60200:
	IF NOT Robot._DI1.Done THEN
		IF _bTargetIsA THEN
			Robot.M_StartMoveBoxToRoundBelt_ClampA(
				CarrierSelect := Info.ClampA_Setting.RoundBeltSetting.ReloadCarrier,
				A2_Sensor := A2_Sensor, A3_Sensor := A3_Sensor,
				RoundBeltSafe := CarrierReady_1st);
		ELSE
			Robot.M_StartMoveBoxToRoundBelt_ClampB(
				CarrierSelect := Info.ClampB_Setting.RoundBeltSetting.ReloadCarrier,
				A2_Sensor := A2_Sensor, A3_Sensor := A3_Sensor,
				RoundBeltSafe := CarrierReady_1st);
		END_IF
	ELSE
		// 圓帶放盒不記數 (非倉儲操作)
		tonTimeOut.IN := FALSE;
		uiExecutingStep := 60300;
	END_IF
	tonTimeOut.IN := TRUE;
	IF tonTimeOut.Q THEN uiResumeStep := 60200; _Abort := TRUE; tonTimeOut.IN := FALSE; END_IF

60300:
	// 釋放圓帶資源 + 清除手臂命令 → 三路分派:
	// 1. buffer > 0: 先去 90000 逆序還原 buffer 盒子 (還原完再由 90010 判斷跳轉)
	// 2. _nAfterPlaceStep > 0: C3/C4 的下一輪入口 (如 3250/3350)
	// 3. 否則: 99000 全部完成
	DAS_CoreSys.MachineControl.fbAllocateArea.M_ResetReloadRoundBeltAction();
	DAS_CoreSys.MachineControl.fbAllocateArea.M_ReleaseRoundBeltAccess(ControlAccess := E_RoundBeltControlAccess.FanucRobot);
	Robot.M_ResetAllCommand();
	IF NOT Robot._DI1.Done THEN
		IF _nBufferCount > 0 THEN
			uiExecutingStep := 90000;
		ELSIF _nAfterPlaceStep > 0 THEN
			uiExecutingStep := _nAfterPlaceStep;
			_nAfterPlaceStep := 0;
		ELSE
			uiExecutingStep := 99000;
		END_IF
	END_IF

// ========== 80000: 雙爪放盒到圓帶 (A 爪先放, B 爪後放) ==========
// 80000: 清除命令 + 立即進入圓帶流程 (不等手臂空閒，並行啟動)
// 81000: 雙爪放圓帶主迴圈 (子步序 uiPlaceBothStep):
//   0:  取得圓帶存取權
//   10: 移動圓帶到 A 爪站位 → 等待到位
//   11: 等待 A 爪載具 sensor 確認 (A2/A3) → 再次取得圓帶存取權
//   20: 等待 Robot Notification (A 爪放完) → Reset 圓帶動作
//   30: 移動圓帶到 B 爪站位
//   40: 等待 B 爪載具到位
//   99: 等待手臂完成
// 81080: 釋放圓帶存取權 + 清除命令 → buffer 還原或完成
80000:
	// 圓帶先動 — 不等手臂完全空閒，手臂清除與圓帶移動並行
	WareHouse.M_ResetReloadBox();
	Robot.M_ResetAllCommand();
	uiExecutingStep := 81000;

81000:
	// ── 子步序: 圓帶側與手臂側並行協調 ──
	// 圓帶側 (uiPlaceBothStep): 依序移到 A站位→確認載具→等A放完→移到 B站位→確認載具
	// 手臂側 (下方 M_StartMoveBoxToRoundBelt_Both): 每 cycle 持續呼叫，根據 CarrierReady 旗標推進
	CASE uiPlaceBothStep OF
	0:
		// 初始化: 取得圓帶控制權，立即開始移動
		CarrierReady_1st := FALSE;
		CarrierReady_2nd := FALSE;
		DAS_CoreSys.MachineControl.fbAllocateArea.M_GetRoundBeltAccess(ControlAccess := E_RoundBeltControlAccess.FanucRobot);
		uiPlaceBothStep := 10;
	10:
		// 圓帶移到 A 爪站位，等待到位 (與手臂清除並行)
		DAS_CoreSys.MachineControl.fbAllocateArea.M_StartReloadRoundBeltAtion(ReloadStation := Info.ClampA_Setting.RoundBeltSetting.Station);
		IF RoundBelt.xDone THEN
			DAS_CoreSys.MachineControl.fbAllocateArea.M_ResetReloadRoundBeltAction();
			DAS_CoreSys.MachineControl.fbAllocateArea.M_ReleaseRoundBeltAccess(ControlAccess := E_RoundBeltControlAccess.FanucRobot);
			CarrierReady_1st := TRUE;	// → 手臂開始 A 爪放盒
			uiPlaceBothStep := 11;
		END_IF
		IF RoundBelt.xError THEN
			_Error := TRUE;
			DAS_CoreSys.MachineControl.fbAllocateArea.M_ResetReloadRoundBeltAction();
			strStatus := 'FB_WareHouseInnerPickToRoundBelt Step 81000: RoundBelt error';
		END_IF
	11:
		// 等待 A 爪對應的載具 sensor 偵測到位 (確認載具已在手臂放盒範圍內)
		// A2 載具用 A2_Sensor 確認, A3 載具用 A3_Sensor 確認
		IF ((Info.ClampA_Setting.RoundBeltSetting.ReloadCarrier = E_ReloadRoundBelt_PlaceAddress.A2) AND A2_Sensor) OR
			((Info.ClampA_Setting.RoundBeltSetting.ReloadCarrier = E_ReloadRoundBelt_PlaceAddress.A3) AND A3_Sensor) THEN
			// 載具到位 → 重新取得圓帶權限 (step 10 釋放過)，準備等手臂放完後移到 B 站位
			DAS_CoreSys.MachineControl.fbAllocateArea.M_GetRoundBeltAccess(ControlAccess := E_RoundBeltControlAccess.FanucRobot);
			uiPlaceBothStep := 20;
		END_IF
	20:
		// 等待手臂 Notification = A 爪放盒完成信號 (手臂程式中途發出，不等全部結束)
		IF Robot._DI1.Notification THEN
			DAS_CoreSys.MachineControl.fbAllocateArea.M_ResetReloadRoundBeltAction();
			// 確認圓帶不在 Done 狀態 (已被 Reset)，才開始移到 B 站位
			IF NOT RoundBelt.xDone THEN
				uiPlaceBothStep := 30;
			END_IF
		END_IF
	30:
		// 圓帶移到 B 爪站位
		DAS_CoreSys.MachineControl.fbAllocateArea.M_GetRoundBeltAccess(ControlAccess := E_RoundBeltControlAccess.FanucRobot);
		DAS_CoreSys.MachineControl.fbAllocateArea.M_StartReloadRoundBeltAtion(ReloadStation := Info.ClampB_Setting.RoundBeltSetting.Station);
		uiPlaceBothStep := 40;
	40:
		// 等待 B 爪站位到位
		IF RoundBelt.xDone THEN
			DAS_CoreSys.MachineControl.fbAllocateArea.M_ResetReloadRoundBeltAction();
			CarrierReady_2nd := TRUE;	// → 手臂開始 B 爪放盒
			uiPlaceBothStep := 99;
		END_IF
		IF RoundBelt.xError THEN
			_Error := TRUE;
			DAS_CoreSys.MachineControl.fbAllocateArea.M_ResetReloadRoundBeltAction();
			strStatus := 'FB_WareHouseInnerPickToRoundBelt Step 81000: RoundBelt error';
		END_IF
	99: // 圓帶側完成，等待手臂側 Done
	END_CASE

	// 手臂側: 每 cycle 持續呼叫，手臂內部根據 CarrierReady 旗標推進雙爪放盒流程
	IF NOT Robot._DI1.Done THEN
		Robot.M_StartMoveBoxToRoundBelt_Both(
			CarrierSelect_ClampA := Info.ClampA_Setting.RoundBeltSetting.ReloadCarrier,
			CarrierSelect_ClampB := Info.ClampB_Setting.RoundBeltSetting.ReloadCarrier,
			A2_Sensor := A2_Sensor, A3_Sensor := A3_Sensor,
			RoundBeltSafe_1st := CarrierReady_1st,
			RoundBeltSafe_2nd := CarrierReady_2nd);
	ELSE
		// 圓帶放盒不記數 (非倉儲操作)
		tonTimeOut.IN := FALSE;
		uiExecutingStep := 81080;
	END_IF
	tonTimeOut.IN := TRUE;
	IF tonTimeOut.Q THEN uiResumeStep := 81000; _Abort := TRUE; tonTimeOut.IN := FALSE; END_IF

81080:
	DAS_CoreSys.MachineControl.fbAllocateArea.M_ResetReloadRoundBeltAction();
	DAS_CoreSys.MachineControl.fbAllocateArea.M_ReleaseRoundBeltAccess(ControlAccess := E_RoundBeltControlAccess.FanucRobot);
	Robot.M_ResetAllCommand();
	IF NOT Robot._DI1.Done THEN
		IF _nBufferCount > 0 THEN
			uiExecutingStep := 90000;		// 有 buffer 要還原
		ELSIF _nAfterPlaceStep > 0 THEN
			uiExecutingStep := _nAfterPlaceStep;	// C3/C4 跳轉到下一輪
			_nAfterPlaceStep := 0;
		ELSE
			uiExecutingStep := 99000;		// 完成
		END_IF
	END_IF

// ========== 90000: Buffer 盒子逆序還原 ==========
// 將之前搬到 buffer 的盒子，逆序 (後進先出) 放回倉儲
// 雙爪路徑: 一次從 buffer 取兩個 → 依序放回倉儲
// 單爪路徑: 剩一個時用目標爪處理
90000:
	_nBufferStep := _nBufferCount;
	BoxReady_1st := FALSE;
	BoxReady_2nd := FALSE;
	uiExecutingStep := 90005;

90005:
	IF _nBufferStep < 1 THEN
		// buffer 還原完成 → 檢查是否有下一輪跳轉 (C3/C4)
		IF _nAfterPlaceStep > 0 THEN
			uiExecutingStep := _nAfterPlaceStep;
			_nAfterPlaceStep := 0;
		ELSE
			uiExecutingStep := 99000;
		END_IF
	ELSIF _nBufferStep >= 2 THEN
		// 剩 2 個以上: 雙爪一次還原兩個
		uiExecutingStep := 90010;
	ELSE
		// 剩 1 個: 單爪還原
		uiExecutingStep := 90040;
	END_IF

// ===== 雙爪 buffer 還原路徑 =====
// Step 1: 雙爪從 buffer 取兩個盒子
90010:
	IF NOT Robot._DI1.Done THEN
		IF _bTargetIsA THEN
			Robot.M_StartRobotAbsMove(
				GetBox := TRUE, UseClampA := TRUE, UseClampB := TRUE,
				Area := E_RobotArea.BufferArea,
				ClampA_Address := _nBufferStep, ClampB_Address := _nBufferStep - 1,
				BoxReady_1 := TRUE, BoxReady_2 := TRUE);
		ELSE
			Robot.M_StartRobotAbsMove(
				GetBox := TRUE, UseClampA := TRUE, UseClampB := TRUE,
				Area := E_RobotArea.BufferArea,
				ClampA_Address := _nBufferStep - 1, ClampB_Address := _nBufferStep,
				BoxReady_1 := TRUE, BoxReady_2 := TRUE);
		END_IF
	ELSE
		// buffer 取盒不記數 (非倉儲操作)
		tonTimeOut.IN := FALSE;
		uiExecutingStep := 90015;
	END_IF
	tonTimeOut.IN := TRUE;
	IF tonTimeOut.Q THEN uiResumeStep := 90010; _Abort := TRUE; tonTimeOut.IN := FALSE; END_IF

90015:
	Robot.M_ResetAllCommand();
	IF NOT Robot._DI1.Done THEN
		BoxReady_1st := FALSE;
		BoxReady_2nd := FALSE;
		uiExecutingStep := 90020;
	END_IF

// Step 2: 目標爪放回倉儲 (buffer 高位, LIFO 先還原)
90020:
	IF NOT Robot._DI1.Done THEN
		IF _bTargetIsA THEN
			WareHouse.M_StartFeedInBox(WareHouseSelect := _wsA, WarehouseCoordinates := _coordsA);
			IF WareHouse.bFeedInBox_Completed THEN BoxReady_1st := TRUE; END_IF
			Robot.M_StartWareHousePlaceBox_ClampA(WareHouseSelect := _wsA, Info := _coordsA, BoxReady_1st := BoxReady_1st);
		ELSE
			WareHouse.M_StartFeedInBox(WareHouseSelect := _wsB, WarehouseCoordinates := _coordsB);
			IF WareHouse.bFeedInBox_Completed THEN BoxReady_2nd := TRUE; END_IF
			Robot.M_StartWareHousePlaceBox_ClampB(WareHouseSelect := _wsB, Info := _coordsB, BoxReady_2nd := BoxReady_2nd);
		END_IF
	ELSE
		// Place 完成通知: 目標爪放回倉儲 (buffer 高位)
		IF ActionIndex < 40 THEN
			IF _bTargetIsA THEN
				ActionRecords[ActionIndex].WareHouse := _wsA; ActionRecords[ActionIndex].Layer := _coordsA.Layer; ActionRecords[ActionIndex].Slide := _coordsA.Slide; ActionRecords[ActionIndex].Clamp := 0;
			ELSE
				ActionRecords[ActionIndex].WareHouse := _wsB; ActionRecords[ActionIndex].Layer := _coordsB.Layer; ActionRecords[ActionIndex].Slide := _coordsB.Slide; ActionRecords[ActionIndex].Clamp := 1;
			END_IF
			ActionRecords[ActionIndex].IsPick := FALSE;
			ActionIndex := ActionIndex + 1;
		END_IF
		tonTimeOut.IN := FALSE;
		uiExecutingStep := 90025;
	END_IF
	tonTimeOut.IN := TRUE;
	IF tonTimeOut.Q THEN uiResumeStep := 90020; _Abort := TRUE; tonTimeOut.IN := FALSE; END_IF

90025:
	Robot.M_ResetAllCommand();
	WareHouse.M_ResetFeedInBox();
	IF NOT Robot._DI1.Done THEN
		BoxReady_1st := FALSE;
		BoxReady_2nd := FALSE;
		uiExecutingStep := 90030;
	END_IF

// Step 3: 協助爪放回倉儲 (buffer 低位)
90030:
	IF NOT Robot._DI1.Done THEN
		IF _bTargetIsA THEN
			WareHouse.M_StartFeedInBox(WareHouseSelect := _wsA, WarehouseCoordinates := _coordsA);
			IF WareHouse.bFeedInBox_Completed THEN BoxReady_2nd := TRUE; END_IF
			Robot.M_StartWareHousePlaceBox_ClampB(WareHouseSelect := _wsA, Info := _coordsA, BoxReady_2nd := BoxReady_2nd);
		ELSE
			WareHouse.M_StartFeedInBox(WareHouseSelect := _wsB, WarehouseCoordinates := _coordsB);
			IF WareHouse.bFeedInBox_Completed THEN BoxReady_1st := TRUE; END_IF
			Robot.M_StartWareHousePlaceBox_ClampA(WareHouseSelect := _wsB, Info := _coordsB, BoxReady_1st := BoxReady_1st);
		END_IF
	ELSE
		// Place 完成通知: 協助爪放回倉儲 (buffer 低位)
		IF ActionIndex < 40 THEN
			IF _bTargetIsA THEN
				ActionRecords[ActionIndex].WareHouse := _wsA; ActionRecords[ActionIndex].Layer := _coordsA.Layer; ActionRecords[ActionIndex].Slide := _coordsA.Slide; ActionRecords[ActionIndex].Clamp := 1;
			ELSE
				ActionRecords[ActionIndex].WareHouse := _wsB; ActionRecords[ActionIndex].Layer := _coordsB.Layer; ActionRecords[ActionIndex].Slide := _coordsB.Slide; ActionRecords[ActionIndex].Clamp := 0;
			END_IF
			ActionRecords[ActionIndex].IsPick := FALSE;
			ActionIndex := ActionIndex + 1;
		END_IF
		tonTimeOut.IN := FALSE;
		uiExecutingStep := 90035;
	END_IF
	tonTimeOut.IN := TRUE;
	IF tonTimeOut.Q THEN uiResumeStep := 90030; _Abort := TRUE; tonTimeOut.IN := FALSE; END_IF

90035:
	Robot.M_ResetAllCommand();
	WareHouse.M_ResetFeedInBox();
	IF NOT Robot._DI1.Done THEN
		BoxReady_1st := FALSE;
		BoxReady_2nd := FALSE;
		_nBufferStep := _nBufferStep - 2;
		uiExecutingStep := 90005;
	END_IF

// ===== 單爪 buffer 還原路徑 (剩一個) =====
90040:
	IF NOT Robot._DI1.Done THEN
		IF _bTargetIsA THEN
			Robot.M_StartRobotAbsMove(
				GetBox := TRUE, UseClampA := TRUE, UseClampB := FALSE,
				Area := E_RobotArea.BufferArea,
				ClampA_Address := _nBufferStep, ClampB_Address := 0,
				BoxReady_1 := TRUE, BoxReady_2 := FALSE);
		ELSE
			Robot.M_StartRobotAbsMove(
				GetBox := TRUE, UseClampA := FALSE, UseClampB := TRUE,
				Area := E_RobotArea.BufferArea,
				ClampA_Address := 0, ClampB_Address := _nBufferStep,
				BoxReady_1 := FALSE, BoxReady_2 := TRUE);
		END_IF
	ELSE
		// buffer 取盒不記數 (非倉儲操作)
		tonTimeOut.IN := FALSE;
		uiExecutingStep := 90045;
	END_IF
	tonTimeOut.IN := TRUE;
	IF tonTimeOut.Q THEN uiResumeStep := 90040; _Abort := TRUE; tonTimeOut.IN := FALSE; END_IF

90045:
	Robot.M_ResetAllCommand();
	IF NOT Robot._DI1.Done THEN
		BoxReady_1st := FALSE;
		BoxReady_2nd := FALSE;
		uiExecutingStep := 90050;
	END_IF

90050:
	IF NOT Robot._DI1.Done THEN
		IF _bTargetIsA THEN
			WareHouse.M_StartFeedInBox(WareHouseSelect := _wsA, WarehouseCoordinates := _coordsA);
			IF WareHouse.bFeedInBox_Completed THEN BoxReady_1st := TRUE; END_IF
			Robot.M_StartWareHousePlaceBox_ClampA(WareHouseSelect := _wsA, Info := _coordsA, BoxReady_1st := BoxReady_1st);
		ELSE
			WareHouse.M_StartFeedInBox(WareHouseSelect := _wsB, WarehouseCoordinates := _coordsB);
			IF WareHouse.bFeedInBox_Completed THEN BoxReady_2nd := TRUE; END_IF
			Robot.M_StartWareHousePlaceBox_ClampB(WareHouseSelect := _wsB, Info := _coordsB, BoxReady_2nd := BoxReady_2nd);
		END_IF
	ELSE
		// Place 完成通知: 放回倉儲 (buffer 逆序還原)
		IF ActionIndex < 40 THEN
			IF _bTargetIsA THEN
				ActionRecords[ActionIndex].WareHouse := _wsA; ActionRecords[ActionIndex].Layer := _coordsA.Layer; ActionRecords[ActionIndex].Slide := _coordsA.Slide; ActionRecords[ActionIndex].Clamp := 0;
			ELSE
				ActionRecords[ActionIndex].WareHouse := _wsB; ActionRecords[ActionIndex].Layer := _coordsB.Layer; ActionRecords[ActionIndex].Slide := _coordsB.Slide; ActionRecords[ActionIndex].Clamp := 1;
			END_IF
			ActionRecords[ActionIndex].IsPick := FALSE;
			ActionIndex := ActionIndex + 1;
		END_IF
		tonTimeOut.IN := FALSE;
		uiExecutingStep := 90055;
	END_IF
	tonTimeOut.IN := TRUE;
	IF tonTimeOut.Q THEN uiResumeStep := 90050; _Abort := TRUE; tonTimeOut.IN := FALSE; END_IF

90055:
	Robot.M_ResetAllCommand();
	WareHouse.M_ResetFeedInBox();
	IF NOT Robot._DI1.Done THEN
		BoxReady_1st := FALSE;
		BoxReady_2nd := FALSE;
		_nBufferStep := _nBufferStep - 1;
		uiExecutingStep := 90005;
	END_IF

// ========== 99000: 流程完成 → 等待 C# 讀取動作紀錄 ==========
99000:
	DAS_CoreSys.MachineControl.fbAllocateArea.M_ResetReloadRoundBeltAction();
	DAS_CoreSys.MachineControl.fbAllocateArea.M_ReleaseRoundBeltAccess(ControlAccess := E_RoundBeltControlAccess.FanucRobot);
	FeedBack := TRUE;
	uiExecutingStep := 99100;

// Step 99100: 等待 C# 確認讀取完成 (5 秒逾時保護)
99100:
	//tonReadComplete(IN := TRUE, PT := T#15S);
	tonReadComplete.IN := true;
	IF ReadComplete THEN
		FeedBack := FALSE;
		tonReadComplete.IN := FALSE;
		Status := 'FB_WareHouseInnerPickToRoundBelt Step 99100: Process completed';
		_Executed := TRUE;
	ELSIF tonReadComplete.Q THEN
		// C# 讀取逾時 → Abort + 設 resume 回 99100，Reset 後可續做
		tonReadComplete.IN := FALSE;
		strStatus := 'FB_WareHouseInnerPickToRoundBelt Step 99100: ReadComplete timeout (C# did not respond within 5s)';
		_UniqueErrorCode := 'E_READ_COMPLETE_TIMEOUT';
		uiResumeStep := 99100;
		_Abort := TRUE;
	END_IF

END_CASE

// 狀態轉換判斷 (每 cycle 在 CASE 之後檢查)
// 優先順序: 完成 > 外部取消 > 中止(逾時) > 錯誤
// _Executed: 由 step 99000 設定，需等 Robot.Halt 解除才實際轉換 (避免手臂急停中換狀態)
// NOT Execute: 外部 (Batch FB 或 HMI) 取消 Execute，直接進入 RESETTING
// _Abort: 由逾時或內部異常設定，進入 ABORTING 清理手臂/倉儲資源
// _Error: 由命令驗證失敗或圓帶錯誤設定，進入 STATE_ERROR 顯示錯誤
IF _Executed AND NOT Robot.Halt THEN
	eState := STATE_DONE;
ELSIF NOT Execute THEN
	eState := STATE_RESETTING;
ELSIF Abort OR _Abort THEN
	eState := STATE_ABORTING;
ELSIF _Error THEN
	eState := STATE_ERROR;
END_IF
END_METHOD

// 重置狀態 — 釋放所有資源 (圓帶/倉儲/手臂)，清除爪動作旗標
// 如果有恢復旗標 (_bRetry)，回到 STATE_EXECUTING 的中斷步序
METHOD M_STATE_RESETTING
VAR_INPUT
END_VAR
// Done := false 更改到Dormant 清除確保，上位檢查到done 後可以直接下Execute

CASE uiResettingStep OF
0:
	// 清除動作紀錄 + 握手旗標
	MEMSET(ADR(ActionRecords), 0, SIZEOF(ActionRecords));
	ActionIndex := 0;
	FeedBack := FALSE;

	// 釋放所有外部資源 → 圓帶/倉儲/手臂回到初始狀態
	DAS_CoreSys.MachineControl.fbAllocateArea.M_ResetReloadRoundBeltAction();
	DAS_CoreSys.MachineControl.fbAllocateArea.M_ReleaseRoundBeltAccess(ControlAccess := E_RoundBeltControlAccess.FanucRobot);
	WareHouse.M_ResetReloadBox();
	WareHouse.M_ResetFeedInBox();
	Robot.M_ResetAllCommand();

	// 清除內部狀態
	tonTimeOut.IN := FALSE;
	tonReadComplete.IN := FALSE;
	strStatus := '';
	_UniqueErrorCode := '0';

//	IF _bRetry THEN
//		_bRetry := FALSE;
//		eState := STATE_EXECUTING;
//		RETURN;
//	END_IF
	uiResettingStep := 100;
100:
//	Done := FALSE;
//	Busy := FALSE;
	_ResetCompleted := TRUE;
END_CASE

IF _ResetCompleted THEN
	eState := STATE_DORMANT;
END_IF
END_METHOD

END_FUNCTION_BLOCK

// ---- Library/20_MachineUnits/21_StorageArea/Service_Robot/FB_WareHouseInnerPickToRoundBeltBatch.TcPOU
// ═══════════════════════════════════════════════════════════════════════════
// FB_WareHouseInnerPickToRoundBeltBatch
// 倉儲內層取盒放圓帶 — 批次服務 FB
// ═══════════════════════════════════════════════════════════════════════════
//
// 【用途】
// 管理最多 40 筆「從倉儲內層取盒放上圓帶」流程,每筆由 FB_WareHouseInnerPickToRoundBelt
// 逐筆執行。批次流程由 C# HMI 透過 ADS 寫入 BatchInfo 結構觸發,PLC 端負責
// 驗證資料、迭代處理、handshake 同步動作紀錄給 C#。
//
// 【設計模式】
// 參照 FB_AllocateMoveAutoBatchMode,以「單筆 FB 內嵌 + 批次迭代」架構:
//   1. 收到 Execute → 驗證整批資料安全 (M_ValidateBatchData)
//   2. 迭代 FlowInfo[0..NrOfFlow-1]
//   3. 跳過無效項 (ID = -1 或 A/B 爪皆 NoWork)
//   4. 對每筆有效流程配置並啟動 fbSingleFlow,等其完成/失敗
//   5. 完成後記錄 WorkedID 供 HMI/C# 回報
//   6. 跨迭代 handshake 清理,確保 C# 看到每筆 FeedBack 上升緣
//
// 【FeedBack / ReadComplete 握手協定】(關鍵,跨迭代正確性依賴)
// 每筆 fbSingleFlow 完成時:
//   PLC:   step 99000 → FeedBack := TRUE (通知 C# 陣列可讀)
//   C#:    收到 FeedBack=TRUE → 讀 ActionRecords → set ReadComplete=TRUE
//   PLC:   step 99100 看 ReadComplete=TRUE → 清 FeedBack → 進 DONE
//   C#:    應在看到 FeedBack=FALSE 時清 ReadComplete=FALSE (維持協定)
// 本 Batch FB 為了防 C# 忘記清 ReadComplete 造成下一迭代 skip handshake,
// 在 Step 100 (新迭代開始) 與 Step 300 (迭代結束) 強制清 BatchInfo.ReadComplete。
//
// 【資料安全約束】
// M_ValidateBatchData 在 Step 0 首次進入時呼叫,檢查:
//   - 每個 Work clamp 的 Station 不可為 Undefined
//   - 所有 Work clamp 的 (Station, ReloadCarrier) 不可重複 (同 flow A/B 兩爪也算)
// 違規 → Error + uiResumeStep:=0 (不可續做,需 C# 修正資料重來)
//
// 【Resume / Pause】
// Resume: 錯誤/逾時後 C# 按 Reset → RESETTING 等 fbSingleFlow 回 DORMANT
//         → 若 _bRetry 直接回 EXECUTING 從 uiResumeStep 繼續
//         uiResumeStep 映射固定為 100 (重新配置+啟動 fbSingleFlow),因 abort
//         過程會清掉 fbSingleFlow 內部狀態,不能回原 step 200
// Pause:  僅在「迭代邊界」生效 (step 0 或 310),不中斷單筆流程
//         危險區段 (100~300) 繼續跑到下個邊界才凍結
//
// Create Date : 2026/04/01
// Owner       : Copilot
// ═══════════════════════════════════════════════════════════════════════════

FUNCTION_BLOCK FB_WareHouseInnerPickToRoundBeltBatch EXTENDS FB_ObjectBase_V2 IMPLEMENTS IBasicElement

VAR_INPUT
	// ----- 外部資源參照 (由上層 FB_StorageArea 綁定) -----
	Robot			: REFERENCE TO FB_FanucRobot_Basic_V2;	// 倉儲區 Fanuc 手臂 (取放動作執行者)
	RoundBelt		: REFERENCE TO FB_RoundBeltService;		// 圓帶服務 (目的地,換區偵測)
	WareHouse		: REFERENCE TO FB_WareHouse;				// 倉儲 FB (ReloadBox / FeedInBox)
	Input			: ST_InputTable;						// IO 輸入表 (sensor 等)

	// ----- 批次資料 (C# HMI ↔ PLC 介面) -----
	// BatchInfo 由 C# 透過 ADS 寫入;PLC 讀 FlowInfo[] 並回寫 WorkedID / ActionRecords
	BatchInfo		: REFERENCE TO ST_WareHouseInnerPickBatch;

	Stop			: BOOL;									// 外部停止信號 (DORMANT 時阻擋 Execute 觸發)
END_VAR

VAR_OUTPUT
	// 無額外 output — 完成/錯誤/忙碌狀態透過 BatchInfo.HandShake 回傳 C#
END_VAR

VAR
	// ----- 狀態與錯誤追蹤 -----
	strStatus			: STRING;			// 當前狀態/錯誤描述 (顯示給 HMI)
	tonTimeOut			: TON;				// Per-iteration 逾時計時器 (PT=600s, step 310 推進時重置)
	_UniqueErrorCode	: STRING;			// 錯誤代碼 (E_NOT_AUTO_MODE / E_BATCH_TIMEOUT / E_FLOW_FAILED /
											// E_STATION_UNDEFINED / E_DUPLICATE_TARGET)
	uiResumeStep		: UDINT := 0;		// 續做點步序 (0 = 不可續做, 其他 = RESETTING retry 回此 step)
	_bRetry				: BOOL;				// 續做旗標 (ABORTED → RESETTING → EXECUTING 路徑標記)

	// ----- 批次迭代控制 -----
	iProcessingIndex	: INT := 0;		// 當前處理的流程索引 (0..NrOfFlow-1)
										// 注意: 續做時保留不歸零 (僅 DORMANT 清),保證從中斷點繼續
	CurrentFlow			: ST_WareHouseInnerPickFlowInfo;	// 當前流程資料快取 (避免 C# 改寫中讀取)

	// ----- 內嵌單筆 FB -----
	// 每筆流程都透過這個實例執行;Step 100 配置參照+啟動,Step 310 等其回到 DORMANT
	fbSingleFlow		: FB_WareHouseInnerPickToRoundBelt;
	_bSingleFlowStarted	: BOOL;		// 追蹤 fbSingleFlow 是否有待清理的執行狀態 (用於 ABORTING)
END_VAR

// ============================================================
// 執行順序: input piping → A00 → A10 → output piping
// 讓 state machine 內的 fbSingleFlow() 看到當前 scan 的 C# 輸入
// (ReadComplete),避免 1 scan 延遲
// ============================================================

// 1. Input piping: C# → fbSingleFlow (在 state machine 前)
IF __ISVALIDREF(BatchInfo) THEN
	fbSingleFlow.ReadComplete := BatchInfo.ReadComplete;
	Execute := BatchInfo.HandShake.Execute;
	Reset	:=BatchInfo.HandShake.Reset ;
END_IF

// 2. Timer PT setup
A00_BasicUnits();

// 3. State machine (含 fbSingleFlow() 呼叫)
SUPER^.A10_StateControl();

// 4. Output piping: fbSingleFlow → C#
IF __ISVALIDREF(BatchInfo) THEN
	BatchInfo.ActionRecords := fbSingleFlow.ActionRecords;
	BatchInfo.ActionIndex := fbSingleFlow.ActionIndex;
	BatchInfo.FeedBack := fbSingleFlow.FeedBack;
	BatchInfo.HandShake.Done := Done;
	BatchInfo.HandShake.Busy := Busy;
	BatchInfo.HandShake.Error := Error;
END_IF
fbSingleFlow (Input := Input);

ACTION A00_BasicUnits:
// 每單筆流程上限 (per-iteration timeout,由 EXECUTING step 310 重置)
// 最多 40 筆 x 600s 單筆 = 6.7hr 批次上限足夠
tonTimeOut(PT := T#900S);
END_ACTION

// 尋找下一筆有效流程
// 從 iProcessingIndex 開始往後掃描 BatchInfo.FlowInfo[]
// 有效條件: ID <> -1 且至少一爪為 Work
// 無效流程自動跳過並記錄 WorkedID
// 回傳 TRUE = 找到有效流程 (iProcessingIndex 已更新), FALSE = 全部完成
METHOD M_FindNextValidFlow : BOOL
VAR_INPUT
END_VAR
VAR
	i		: INT;
	bValid	: BOOL;
END_VAR
IF NOT __ISVALIDREF(BatchInfo) THEN
	M_FindNextValidFlow := FALSE;
	RETURN;
END_IF

IF BatchInfo.NrOfFlow = 0 THEN
	M_FindNextValidFlow := FALSE;
	RETURN;
END_IF

FOR i := iProcessingIndex TO UINT_TO_INT(BatchInfo.NrOfFlow) - 1 BY 1 DO
	bValid := FALSE;

	// 檢查 flow 是否有效 (ID 不為 -1)
	IF BatchInfo.FlowInfo[i].ID <> -1 THEN
		// 檢查是否至少一爪有 Work 行為
		IF BatchInfo.FlowInfo[i].ClampA_Setting.Behavior = E_ClampWork.Work
		OR BatchInfo.FlowInfo[i].ClampB_Setting.Behavior = E_ClampWork.Work THEN
			bValid := TRUE;
		END_IF
	END_IF

	IF bValid THEN
		iProcessingIndex := i;
		CurrentFlow := BatchInfo.FlowInfo[i];
		M_FindNextValidFlow := TRUE;
		RETURN;
	ELSE
		// 標記跳過的 flow 為已處理
		BatchInfo.WorkedID[i] := BatchInfo.FlowInfo[i].ID;
	END_IF
END_FOR

// 沒有更多有效流程
M_FindNextValidFlow := FALSE;
END_METHOD

// ───────────────────────────────────────────────────────────
// M_STATE_ABORTED — 已中止 (可續做錯誤)
// ───────────────────────────────────────────────────────────
// 進入條件:
//   M_STATE_ABORTING 完成清理 (_AbortCompleted=TRUE) 後進入
//
// 特性:
//   - 顯示 Aborted=TRUE + Error=TRUE + strStatus
//   - 等待 C# 透過 BatchInfo.HandShake.Reset 觸發續做或重來
//
// Reset 行為:
//   - uiResumeStep > 0 → 設 _bRetry, uiExecutingStep := uiResumeStep
//                        RESETTING 會等 fbSingleFlow 回 DORMANT 後直接跳 EXECUTING
//                        (從中斷點續做,保留 iProcessingIndex)
//   - uiResumeStep = 0 → 單純 RESETTING → DORMANT,下次 Execute 從頭跑
METHOD M_STATE_ABORTED
VAR_INPUT
END_VAR
IF NOT _bRetry THEN
	Busy 	:= FALSE;
	Aborted := TRUE;
	Error 	:= TRUE;
	Status 	:= strStatus;
	_AbortCompleted := FALSE;
	uiAbortingStep  := 0;
END_IF
// 判斷內部Serivce 已經在aborted 狀態等著才能讓 FB reset
IF fbSingleFlow.eState = STATE_Aborted THEN
	IF reset THEN
		fbSingleFlow();
		fbSingleFlow.Reset := TRUE;

		_bRetry := TRUE;
		Aborted	:= FALSE;
		Error	:= FALSE;
	END_IF
END_IF

// 狀態機切換
IF NOT Execute THEN
	eState := STATE_RESETTING;
ELSIF Execute AND _bRetry THEN
	IF fbSingleFlow.eState = STATE_EXECUTING THEN
		fbSingleFlow.Reset := FALSE;
		IF uiResumeStep > 0 THEN
			status			:= '';
			uiExecutingStep := uiResumeStep;
			eState 			:= STATE_EXECUTING;
		END_IF
	END_IF
END_IF
END_METHOD

// ───────────────────────────────────────────────────────────
// M_STATE_ABORTING — 中止流程
// ───────────────────────────────────────────────────────────
// 職責:
//   把正在執行的 fbSingleFlow 中止,等其自身 ABORTING → ABORTED
//   跑完後設 _AbortCompleted 進入 STATE_ABORTED。
//   fbSingleFlow 的 ABORTING 內部會處理 Robot/WareHouse/RoundBelt 的資源釋放。
//
// 進入條件:
//   M_STATE_EXECUTING 設 _Abort := TRUE 時觸發
//   (timeout, 單筆流程失敗, Auto mode 脫離等)
//
// 步序:
//   0:    若 _bSingleFlowStarted=TRUE → 發送 fbSingleFlow.Abort := TRUE, 跳 100
//         (若單筆 FB 尚未啟動過,直接跳 9999 略過等待)
//   100:  每 cycle 呼叫 fbSingleFlow() 推進其內部中止狀態機
//         等待條件 (任一滿足): 未啟動 / fbSingleFlow.Aborted / fbSingleFlow 不忙碌
//         → 清 fbSingleFlow.Abort := FALSE, 跳 9999
//   9999: _AbortCompleted := TRUE → base class 轉入 STATE_ABORTED
//
// 注意:
//   iProcessingIndex 不在此清除 (保留供續做),由 DORMANT 才清
METHOD M_STATE_ABORTING
VAR_INPUT
END_VAR
CASE uiAbortingStep OF
0:
	_Abort:= FALSE;
	_bRetry := false;
	// Abort single-flow FB if running
	IF _bSingleFlowStarted THEN
		fbSingleFlow.Abort := TRUE;
		fbSingleFlow();
	END_IF
	uiAbortingStep := 100;

100:
	// 每 cycle 呼叫 fbSingleFlow() 推進其內部中止狀態機 (ABORTING → ABORTED)
	// 等待條件: 未啟動 / 已中止 / 不在忙碌 → 任一滿足即視為中止完成
	fbSingleFlow();
	IF fbSingleFlow.Aborted OR NOT fbSingleFlow.Busy THEN
		fbSingleFlow.Abort := FALSE;
		uiAbortingStep := 9999;
	END_IF

9999:
	_AbortCompleted := TRUE;
END_CASE

IF NOT Execute THEN
	eState := STATE_RESETTING;
ELSIF Execute AND _AbortCompleted THEN
	eState := STATE_Aborted;
END_IF
END_METHOD

// ───────────────────────────────────────────────────────────
// M_STATE_DONE — 批次完成等待
// ───────────────────────────────────────────────────────────
// 批次全部流程成功完成後進入此狀態,設 Done=TRUE 讓 C# 收到完成回報。
// 等 C# 清 BatchInfo.HandShake.Execute (表示收到完成訊號) 後轉 RESETTING。
METHOD M_STATE_DONE
VAR_INPUT
END_VAR
Busy   := FALSE;
_Error := Error := FALSE;
_Abort := Abort := FALSE;
Done   := TRUE;

IF __ISVALIDREF(BatchInfo) THEN
	IF NOT BatchInfo.HandShake.Execute THEN
		eState := STATE_RESETTING;
	END_IF
ELSIF NOT Execute THEN
	eState := STATE_RESETTING;
END_IF
END_METHOD

// ───────────────────────────────────────────────────────────
// M_STATE_DORMANT — 休眠 / 靜止就緒狀態
// ───────────────────────────────────────────────────────────
// 職責:
//   1. 每 scan 重置所有 FB-level 輸出旗標與內部狀態至乾淨初值
//   2. 清除上一輪殘留的 BatchInfo.WorkedID (避免 C# 誤讀舊資料)
//   3. 監聽 BatchInfo.HandShake.Execute / Reset 握手信號
//
// 進入條件:
//   - 從 M_STATE_RESETTING 完成時進入
//   - 首次上電時的初始狀態
//
// 離開條件:
//   - BatchInfo.HandShake.Execute=TRUE AND NOT Stop → STATE_EXECUTING
//
// 備註:
//   每 scan 都跑 (PLC 狀態機性質),所以所有 reset 都必須冪等。
//   M_RecoveryAllObjects 不放這裡,因 fbSingleFlow 的清理由 RESETTING 處理。
METHOD M_STATE_DORMANT
VAR_INPUT
END_VAR
// 清除所有輸出與內部狀態
Busy				:= FALSE;
Done				:= FALSE;
Aborted				:= FALSE;
Error				:= FALSE;
ErrorID				:= 0;
Status				:= '';
_ResetCompleted		:= FALSE;
_Error				:= FALSE;
_Executed			:= FALSE;
_Abort				:= FALSE;
uiExecutingStep		:= 0;
uiResettingStep		:= 0;
uiResumeStep		:= 0;
uiAbortingStep		:= 0;

tonTimeOut.IN		:= FALSE;
_UniqueErrorCode	:= '0';

// 清除批次狀態
iProcessingIndex	:= 0;
_bSingleFlowStarted	:= FALSE;

// 清除上一輪殘留的 WorkedID (避免 C# 誤讀舊資料)
IF __ISVALIDREF(BatchInfo) THEN
	MEMSET(ADR(BatchInfo.WorkedID), 0, SIZEOF(BatchInfo.WorkedID));
END_IF

_AbortCompleted		:= FALSE;
_bRetry				:= FALSE;

// 監聽 HMI/C# 透過 ADS 寫入的 HandShake 信號
// Execute: C# 設定 BatchInfo.HandShake.Execute = TRUE 觸發批次開始
// Reset: C# 在 Error/Aborted 後設定 Reset 清除狀態 (若有 uiResumeStep 則恢復)
IF __ISVALIDREF(BatchInfo) THEN
	IF BatchInfo.HandShake.Execute AND NOT Stop THEN
		Execute := TRUE;
		eState := STATE_EXECUTING;
	END_IF

	IF BatchInfo.HandShake.Reset THEN
		Reset := TRUE;
	END_IF
END_IF
END_METHOD

// ───────────────────────────────────────────────────────────
// M_STATE_ERROR — 不可續做錯誤顯示
// ───────────────────────────────────────────────────────────
// 進入條件:
//   M_STATE_EXECUTING 設 _Error := TRUE (資料驗證失敗等)
//
// 特性:
//   - 此狀態代表「不可續做」,必須 C# 修正資料後從頭重來
//   - 可續做錯誤 (timeout / 單筆失敗) 走 STATE_ABORTING → STATE_ABORTED 路徑
//   - 等 C# 清 BatchInfo.HandShake.Execute 後進 RESETTING
METHOD M_STATE_ERROR
VAR_INPUT
END_VAR
Busy := FALSE;
Error := TRUE;
Status := strStatus;

IF NOT Execute THEN
	eState := STATE_RESETTING;
END_IF
END_METHOD

// ═══════════════════════════════════════════════════════════════════════════
// M_STATE_EXECUTING — 批次迭代執行主狀態
// ═══════════════════════════════════════════════════════════════════════════
//
// 【進入條件】
//   M_STATE_DORMANT 看到 BatchInfo.HandShake.Execute=TRUE AND NOT Stop 後轉入
//
// 【每 cycle 前置檢查】(在 CASE 之前執行)
//   A. Auto mode 檢查: 若不在 Auto → _Abort (避免軸控衝突)
//   B. Pause gate: 僅在 step 0 / 310 (迭代邊界) 生效
//                 危險區段 (100~300) 繼續跑到下個邊界才凍結
//   C. Per-iteration timeout (600s): 超時 → _Abort, uiResumeStep := 100
//
// 【步序總覽】
//   0:      首次進入: M_ValidateBatchData() 整批驗證 (Station 不為 Undefined, 無重複目的地)
//           驗證失敗 → _Error + uiResumeStep:=0 (不可續做)
//           M_FindNextValidFlow(): 從 iProcessingIndex 掃描下一筆有效 flow
//           → 無: 跳 99000 (全部完成)
//           → 找到: 快取 CurrentFlow, 跳 100
//
//   100:    新迭代起始 — 強制清 handshake 狀態 (BatchInfo.FeedBack/ReadComplete + fbSingleFlow.ReadComplete)
//           確保 C# 一定看到本迭代的 FeedBack 上升緣,不被上一迭代的殘留 ack 誤判
//           配置 fbSingleFlow.Robot/RoundBelt/WareHouse/Input/Info/Stop 參照
//           啟動 fbSingleFlow.Execute := TRUE, 跳 200
//
//   200:    等待單筆 FB 完成 — 每 cycle 呼叫 fbSingleFlow() 推進其內部狀態機
//           → fbSingleFlow.Done: 流程成功 → 跳 300
//           → fbSingleFlow.Error/Aborted: 單筆流程失敗 → _Abort,
//             uiResumeStep := 100 (必須回 100 重新配置,因 abort 會清掉 fbSingleFlow 狀態)
//
//   300:    記錄完成 — 寫入 BatchInfo.WorkedID[iProcessingIndex] := CurrentFlow.ID
//           強制清 BatchInfo.ReadComplete (防 C# 遺忘)
//           釋放 fbSingleFlow.Execute := FALSE (讓它進入 RESETTING → DORMANT)
//           跳 310
//
//   310:    等待 fbSingleFlow 完成 RESETTING → DORMANT (Busy/Done/Error 皆 FALSE)
//           避免下一筆配置時與單筆 FB 的清理步序衝突
//           滿足 → iProcessingIndex + 1, 重置 tonTimeOut, 回 0 (處理下一筆)
//
//   99000:  批次全部完成 — _Executed := TRUE → STATE_DONE
//
// 【狀態轉換優先順序】(CASE 後檢查)
//   _Error → STATE_ERROR      (資料驗證失敗等不可續做錯誤)
//   _Abort → STATE_ABORTING   (timeout, 單筆流程失敗等可續做錯誤)
//   _Executed → STATE_DONE    (批次完成)
//
// ═══════════════════════════════════════════════════════════════════════════
METHOD M_STATE_EXECUTING
VAR_INPUT
END_VAR
Busy := TRUE;
tonTimeOut.IN := TRUE;

// 非自動模式直接中止 (避免軸控衝突)
IF GVL_Machine.PackTags[UnitNo.Storage].Status.UnitModeCurrent <> E_UnitMode.Auto THEN
	strStatus := 'FB_WareHouseInnerPickToRoundBeltBatch: Not in Auto mode';
	_UniqueErrorCode := 'E_NOT_AUTO_MODE';
	_Abort := TRUE;
END_IF

// ============================================================
// Pause (Fix P1): 僅在「迭代邊界」生效,避免單筆流程被卡在半途
// 安全 step: 0 (尋找下一筆) / 310 (等 fbSingleFlow 回 DORMANT)
// 危險 step (100~300): 跑完當前這一筆才能凍結
// ============================================================
IF __ISVALIDREF(BatchInfo) AND BatchInfo.Pause THEN
	IF uiExecutingStep = 0 OR uiExecutingStep = 310 THEN
		strStatus := 'FB_WareHouseInnerPickToRoundBeltBatch: Paused (at iteration boundary)';
	END_IF
	// 非安全 step: 繼續跑直到下一個 iteration 邊界
END_IF

// 批次逾時 (per-iteration, step 310 推進時會重置): 單筆上限 600s
// Resume 映射: 無論 timeout 發生在哪個 step,都回 step 100 重新配置 fbSingleFlow
// (abort 過程會清掉 fbSingleFlow 狀態,直接回原 step 沒用)
IF tonTimeOut.Q THEN
	strStatus := 'FB_WareHouseInnerPickToRoundBeltBatch: Batch per-iteration timeout';
	_UniqueErrorCode := 'E_BATCH_TIMEOUT';
	uiResumeStep := 100;
	_Abort := TRUE;
END_IF

CASE uiExecutingStep OF

// ===== Step 0: 資料安全檢查 + 尋找下一筆有效流程 =====
0:
	// 首次進入 (iProcessingIndex=0 且非 retry) 時驗證整個 batch 資料
	// retry 路徑 (_bRetry 由 RESETTING 清) 不重驗,避免重跑時 C# 結構已變
	IF iProcessingIndex = 0 THEN
		IF NOT M_ValidateBatchData() THEN
			// 資料驗證失敗 → 直接報錯,不可續做 (需 C# 修正資料後重來)
			uiResumeStep := 0;
			_Error := TRUE;
		END_IF
	END_IF

	IF NOT M_FindNextValidFlow() THEN
		// 所有流程已處理完畢 → 跳到完成
		uiExecutingStep := 99000;
	ELSE
		strStatus := CONCAT('Processing flow #', INT_TO_STRING(iProcessingIndex));
		uiExecutingStep := 100;
	END_IF

// ===== Step 100: 配置並啟動單筆 FB =====
100:
	// Safety: 新迭代開始,強制清 handshake 狀態,確保 C# 一定看到本迭代的 FeedBack 上升緣
	// 即使 C# 上一迭代忘了清 ReadComplete,也不會被本迭代的 step 99100 誤認為已 ack
	IF __ISVALIDREF(BatchInfo) THEN
		BatchInfo.FeedBack := FALSE;
		BatchInfo.ReadComplete := FALSE;
	END_IF
	fbSingleFlow.ReadComplete := FALSE;

	// 將手臂/圓帶/倉儲參照及當前流程資料傳入 fbSingleFlow
	fbSingleFlow.Robot REF= Robot;
	fbSingleFlow.RoundBelt REF= RoundBelt;
	fbSingleFlow.WareHouse REF= WareHouse;
	fbSingleFlow.Input := Input;
	fbSingleFlow.Info := CurrentFlow;
	fbSingleFlow.Stop := Stop;
	fbSingleFlow.Execute := TRUE;
	_bSingleFlowStarted := TRUE;
	uiExecutingStep := 200;

// ===== Step 200: 等待單筆 FB 完成 =====
200:
	// 每 cycle 呼叫 fbSingleFlow 推進其狀態機
	fbSingleFlow();

	IF fbSingleFlow.Done THEN
		// 流程成功完成 → 記錄並推進
		uiExecutingStep := 300;
	ELSIF fbSingleFlow.Error OR fbSingleFlow.Aborted THEN
		// 流程失敗 → 中止批次
		// Resume 必須回 step 100 重新配置 fbSingleFlow (abort 後 fbSingleFlow 狀態已被清)
		// 不能回 step 200,因為 step 200 假設 fbSingleFlow 已在執行中
		strStatus := CONCAT('Flow #', CONCAT(INT_TO_STRING(iProcessingIndex), ' failed'));
		_UniqueErrorCode := 'E_FLOW_FAILED';
		uiResumeStep := 100;
		_Abort := TRUE;
	END_IF

// ===== Step 300: 記錄完成 + 釋放單筆 FB =====
300:
	// 寫入 WorkedID 供 HMI/C# 回報
	IF __ISVALIDREF(BatchInfo) THEN
		BatchInfo.WorkedID[iProcessingIndex] := CurrentFlow.ID;
		// Safety: 強制清 C# 的 ack,避免殘留 TRUE 讓下一迭代 skip handshake
		BatchInfo.ReadComplete := FALSE;
	END_IF

	// 釋放單筆 FB: Execute := FALSE → 讓它進入 RESETTING → DORMANT
	fbSingleFlow.Execute := FALSE;
	fbSingleFlow();
	_bSingleFlowStarted := FALSE;
	uiExecutingStep := 310;

// ===== Step 310: 等待單筆 FB 回到 DORMANT 後再推進 =====
310:
	// 確保 fbSingleFlow 完成 RESETTING 流程 (MEMSET + 釋放資源)
	// 避免下一筆流程配置時與 RESETTING 步序衝突
	fbSingleFlow();
	IF NOT fbSingleFlow.Busy AND NOT fbSingleFlow.Done AND NOT fbSingleFlow.Error THEN
		iProcessingIndex := iProcessingIndex + 1;
		// Per-iteration timeout reset: 下一筆重新計時 600s
		tonTimeOut.IN := FALSE;
		uiExecutingStep := 0;
	END_IF

// ===== Step 99000: 批次全部完成 =====
99000:
	_Executed := TRUE;

END_CASE

// ===== 狀態切換 (參照 FB_ObjectBase_V2 / FB_AllocateMoveAutoBatchMode 模式) =====
IF __ISVALIDREF(BatchInfo) THEN
	IF NOT BatchInfo.HandShake.Execute THEN
		eState := STATE_RESETTING;
	ELSIF _Error THEN
		eState := STATE_ERROR;
	ELSIF _Abort THEN
		eState := STATE_ABORTING;
	ELSIF _Executed THEN
		eState := STATE_DONE;
	END_IF
END_IF
END_METHOD

// ───────────────────────────────────────────────────────────
// M_STATE_RESETTING — 重置流程 (含續做分流)
// ───────────────────────────────────────────────────────────
// 職責:
//   從 ABORTED/ERROR/DONE 回到 DORMANT (或直接續做回 EXECUTING),
//   並確保 fbSingleFlow 真的走完自己的 RESETTING → DORMANT,避免 race。
//
// 續做 vs 正常 reset 的差別:
//   - 續做 (_bRetry=TRUE): 由 ABORTED state method 收到 Reset 且 uiResumeStep>0 時設旗標,
//     此時 uiExecutingStep 已被寫回 uiResumeStep (通常是 100),步序 50 等 fbSingleFlow
//     真的回 DORMANT 後,直接跳 STATE_EXECUTING,**不經 DORMANT**,
//     所以 iProcessingIndex 保留、從中斷點繼續。
//   - 正常 reset (_bRetry=FALSE): 步序 50 等 fbSingleFlow 回 DORMANT → 步序 100 → DORMANT,
//     DORMANT 會完整清 iProcessingIndex 等狀態,下次 Execute 從頭跑。
//
// 步序:
//   0:    清 Done/Error/Aborted/tonTimeOut.IN, 下 fbSingleFlow.Reset := TRUE 並呼叫一次
//         無條件跳 50 (無論 _bRetry 真假都要等 fbSingleFlow 真的回 DORMANT)
//   50:   每 cycle 呼叫 fbSingleFlow() 推進其 RESETTING,釋放 Reset
//         等待條件: fbSingleFlow 的 Busy/Done/Error/Aborted 全 FALSE
//         滿足後:
//           _bRetry → 清旗標 + STATE_EXECUTING (續做路徑,跳過 100 與 DORMANT)
//           否則    → 跳 100 (正常路徑)
//   100:  _ResetCompleted := TRUE → base class 轉入 STATE_DORMANT
METHOD M_STATE_RESETTING
VAR_INPUT
END_VAR
// Done := false 更改到Dormant 清除確保，上位檢查到done 後可以直接下Execute

CASE uiResettingStep OF
0:
	Error := FALSE;
	Aborted := FALSE;
	tonTimeOut.IN := FALSE;

	// Reset single-flow FB
	//fbSingleFlow.Reset := TRUE;
	fbSingleFlow();
	fbSingleFlow.Execute := FALSE;


	// _bRetry = TRUE: 由 ABORTED 狀態透過 Reset 觸發
	// 無論 retry 或正常 reset,都要先等 fbSingleFlow 真的回到 DORMANT,
	// 避免 fbSingleFlow 還在 RESETTING 時就被 EXECUTING 視為新迭代
	uiResettingStep := 50;

50:
	// 等待 fbSingleFlow 完成 RESETTING → DORMANT (條件: 所有狀態 flag 都 FALSE)
//	fbSingleFlow.Reset := FALSE;
//	fbSingleFlow();
//	IF NOT fbSingleFlow.Busy AND NOT fbSingleFlow.Done AND NOT fbSingleFlow.Error AND NOT fbSingleFlow.Aborted THEN
//		IF _bRetry THEN
//			// 續做路徑: uiExecutingStep 已被設回 uiResumeStep,直接回 EXECUTING
//			_bRetry := FALSE;
//			eState := STATE_EXECUTING;
//			RETURN;
//		END_IF
//		uiResettingStep := 100;
//	END_IF
	fbSingleFlow();
	IF fbSingleFlow.eState = STATE_DORMANT THEN
		uiResettingStep := 100;
	END_IF

100:
//	Done := FALSE;
//	Busy := FALSE;
	_ResetCompleted := TRUE;
END_CASE
IF _ResetCompleted THEN
	eState := STATE_DORMANT;
END_IF
END_METHOD

// 驗證批次資料安全性
// 檢查項目:
//   1. 同一個 (Station, ReloadCarrier) 目的地不能重複出現 (包括同 flow 內 A/B 兩爪)
//   2. 有 Work 的 clamp,其 Station 不能是 Undefined
// 若有任何違規 → 設 Error + strStatus + 回傳 FALSE
// 通過 → 回傳 TRUE
//
// 掃描範圍: BatchInfo.FlowInfo[0..NrOfFlow-1],只檢查 ID<>-1 且 clamp Behavior=Work 的項目
METHOD M_ValidateBatchData : BOOL
VAR_INPUT
END_VAR
VAR
	i, j			: INT;
	nTargets		: INT;					// 已收集的有效目的地數量
	arTargets		: ARRAY[0..79] OF DINT;	// 40 flow x 2 clamp = 80 max. Pack 成 DINT: station*16 + carrier
	nKey			: DINT;
END_VAR
IF NOT __ISVALIDREF(BatchInfo) THEN
	M_ValidateBatchData := FALSE;
	RETURN;
END_IF

nTargets := 0;

FOR i := 0 TO UINT_TO_INT(BatchInfo.NrOfFlow) - 1 BY 1 DO
	IF BatchInfo.FlowInfo[i].ID = -1 THEN
		CONTINUE;
	END_IF

	// ----- A 爪 -----
	IF BatchInfo.FlowInfo[i].ClampA_Setting.Behavior = E_ClampWork.Work THEN
		IF BatchInfo.FlowInfo[i].ClampA_Setting.RoundBeltSetting.Station = E_RoundBeltStation.Undefined THEN
			strStatus := CONCAT('Flow #', CONCAT(INT_TO_STRING(i), ' ClampA Station Undefined'));
			_UniqueErrorCode := 'E_STATION_UNDEFINED';
			M_ValidateBatchData := FALSE;
			RETURN;
		END_IF

		// Pack (Station, ReloadCarrier) → DINT key
		// Station: UINT enum (1..40), Carrier: INT enum (0..4)
		nKey := UINT_TO_DINT(BatchInfo.FlowInfo[i].ClampA_Setting.RoundBeltSetting.Station) * 16
			  + INT_TO_DINT(BatchInfo.FlowInfo[i].ClampA_Setting.RoundBeltSetting.ReloadCarrier);

		// 檢查重複
		FOR j := 0 TO nTargets - 1 BY 1 DO
			IF arTargets[j] = nKey THEN
				strStatus := CONCAT('Duplicate target at flow #', INT_TO_STRING(i));
				_UniqueErrorCode := 'E_DUPLICATE_TARGET';
				M_ValidateBatchData := FALSE;
				RETURN;
			END_IF
		END_FOR
		arTargets[nTargets] := nKey;
		nTargets := nTargets + 1;
	END_IF

	// ----- B 爪 -----
	IF BatchInfo.FlowInfo[i].ClampB_Setting.Behavior = E_ClampWork.Work THEN
		IF BatchInfo.FlowInfo[i].ClampB_Setting.RoundBeltSetting.Station = E_RoundBeltStation.Undefined THEN
			strStatus := CONCAT('Flow #', CONCAT(INT_TO_STRING(i), ' ClampB Station Undefined'));
			_UniqueErrorCode := 'E_STATION_UNDEFINED';
			M_ValidateBatchData := FALSE;
			RETURN;
		END_IF

		nKey := UINT_TO_DINT(BatchInfo.FlowInfo[i].ClampB_Setting.RoundBeltSetting.Station) * 16
			  + INT_TO_DINT(BatchInfo.FlowInfo[i].ClampB_Setting.RoundBeltSetting.ReloadCarrier);

		FOR j := 0 TO nTargets - 1 BY 1 DO
			IF arTargets[j] = nKey THEN
				strStatus := CONCAT('Duplicate target at flow #', INT_TO_STRING(i));
				_UniqueErrorCode := 'E_DUPLICATE_TARGET';
				M_ValidateBatchData := FALSE;
				RETURN;
			END_IF
		END_FOR
		arTargets[nTargets] := nKey;
		nTargets := nTargets + 1;
	END_IF
END_FOR

M_ValidateBatchData := TRUE;
END_METHOD

END_FUNCTION_BLOCK

// ---- Library/20_MachineUnits/21_StorageArea/Service_Robot/FB_FeedInRoundBeltBoxBatch.TcPOU
// ═══════════════════════════════════════════════════════════════════════════
// FB_FeedInRoundBeltBoxBatch
// 圓帶回倉 — 批次服務 FB
// ═══════════════════════════════════════════════════════════════════════════
//
// 【用途】
// 管理最多 40 筆「從圓帶取盒回倉儲 / 或放到 PullOut」流程,每筆由
// FB_FeedInRoundBeltBoxToWareHouse (HandshakeMode=TRUE) 逐筆執行。
// 每筆 flow 可獨立決定目的地: WareHouseA / WareHouseB / PullOutInner / PullOutOuter
//
// 【設計模式】
// 仿 FB_WareHouseInnerPickToRoundBeltBatch:
//   1. 收到 Execute → 迭代 FlowInfo[0..NrOfFlow-1]
//   2. 跳過無效項 (ID = -1 或 A/B 爪皆 NoWork)
//   3. 對每筆有效流程配置並啟動 fbSingleFlow,等其完成/失敗
//   4. 每筆完成後 PLC 透過 FeedBack/ReadComplete 等 C# 讀完 ActionRecords 才進下一筆
//   5. 跨迭代強制清 handshake 防 C# 遺漏
//
// 【FeedBack / ReadComplete 握手協定】
// 同 FB_WareHouseInnerPickToRoundBeltBatch:
//   PLC: 單筆完成 → FeedBack:=TRUE → 等 ReadComplete=TRUE → 清 FeedBack → 進下一筆
//   C#:  看到 FeedBack=TRUE → 讀 ActionRecords → 寫 ReadComplete=TRUE → 等 FeedBack=FALSE → 清 ReadComplete
//
// 【Resume / Pause】
// Resume: 錯誤後 C# 按 Reset → 從 uiResumeStep 繼續 (固定回 100 重新配置 fbSingleFlow)
// Pause:  僅在迭代邊界 (step 0 / 310) 生效, 不中斷單筆流程
//
// Create Date : 2026/04/14
// ═══════════════════════════════════════════════════════════════════════════

FUNCTION_BLOCK FB_FeedInRoundBeltBoxBatch EXTENDS FB_ObjectBase_V2 IMPLEMENTS IBasicElement

VAR_INPUT
	// ----- 外部資源參照 -----
	Robot			: REFERENCE TO FB_FanucRobot_Basic_V2;	// 倉儲區 Fanuc 手臂
	RoundBelt		: REFERENCE TO FB_RoundBeltService;		// 圓帶服務
	WareHouse		: REFERENCE TO FB_WareHouse;				// 倉儲 FB
	Input			: ST_InputTable;						// IO 輸入表

	// ----- 批次資料 (C# HMI ↔ PLC 介面) -----
	BatchInfo		: REFERENCE TO ST_FeedInRBBatch;

	Stop			: BOOL;									// 外部停止信號
END_VAR

VAR_OUTPUT
END_VAR

VAR
	// ----- 狀態與錯誤追蹤 -----
	strStatus			: STRING;
	tonTimeOut			: TON;				// Per-iteration 逾時 (PT=600s, step 310 推進時重置)
	_UniqueErrorCode	: STRING;
	uiResumeStep		: UDINT := 0;
	_bRetry				: BOOL;

	// ----- 批次迭代控制 -----
	iProcessingIndex	: INT := 0;
	CurrentFlow			: ST_FeedInRBFlowInfo;

	// ----- 內嵌單筆 FB -----
	fbSingleFlow		: FB_FeedInRoundBeltBoxToWareHouse;
	_bSingleFlowStarted	: BOOL;
END_VAR

// ============================================================
// 執行順序: input piping → A00 → A10 → output piping
// ============================================================

// 1. Input piping: C# → fbSingleFlow (只轉 ReadComplete,不碰 Execute/Reset)
IF __ISVALIDREF(BatchInfo) THEN
	fbSingleFlow.ReadComplete := BatchInfo.ReadComplete;
	Execute := BatchInfo.HandShake.Execute;
	Reset	:= BatchInfo.HandShake.Reset;
END_IF

// 2. Timer PT setup
A00_BasicUnits();

// 3. State machine
SUPER^.A10_StateControl();

// 4. Output piping: fbSingleFlow → C#
IF __ISVALIDREF(BatchInfo) THEN
	BatchInfo.ActionRecords := fbSingleFlow.ActionRecords;
	BatchInfo.ActionIndex := fbSingleFlow.ActionIndex;
	BatchInfo.FeedBack := fbSingleFlow.FeedBack;
	BatchInfo.HandShake.Done := Done;
	BatchInfo.HandShake.Busy := Busy;
	BatchInfo.HandShake.Error := Error;
END_IF

ACTION A00_BasicUnits:
// Per-iteration timeout, step 310 推進時重置
tonTimeOut(PT := T#600S);
// 每 scan 更新 Input (IO 輸入表),確保 fbSingleFlow 內部讀到最新 sensor
// 只設屬性不呼叫 FB — fbSingleFlow() 呼叫只在 M_STATE_EXECUTING step 200/300/310
fbSingleFlow.Input := Input;
END_ACTION

// 尋找下一筆有效流程
// 從 iProcessingIndex 開始往後掃描 BatchInfo.FlowInfo[]
// 有效條件: ID <> -1 且至少一爪為 Work
// 無效流程自動跳過並記錄 WorkedID
// 回傳 TRUE = 找到有效流程 (iProcessingIndex 已更新), FALSE = 全部完成
METHOD M_FindNextValidFlow : BOOL
VAR_INPUT
END_VAR
VAR
	i		: INT;
	bValid	: BOOL;
END_VAR
IF NOT __ISVALIDREF(BatchInfo) THEN
	M_FindNextValidFlow := FALSE;
	RETURN;
END_IF

IF BatchInfo.NrOfFlow = 0 THEN
	M_FindNextValidFlow := FALSE;
	RETURN;
END_IF

FOR i := iProcessingIndex TO UINT_TO_INT(BatchInfo.NrOfFlow) - 1 BY 1 DO
	bValid := FALSE;

	IF BatchInfo.FlowInfo[i].ID <> -1 THEN
		IF BatchInfo.FlowInfo[i].ClampA_Setting.Behavior = E_ClampWork.Work
		OR BatchInfo.FlowInfo[i].ClampB_Setting.Behavior = E_ClampWork.Work THEN
			bValid := TRUE;
		END_IF
	END_IF

	IF bValid THEN
		iProcessingIndex := i;
		CurrentFlow := BatchInfo.FlowInfo[i];
		M_FindNextValidFlow := TRUE;
		RETURN;
	ELSE
		BatchInfo.WorkedID[i] := BatchInfo.FlowInfo[i].ID;
	END_IF
END_FOR

M_FindNextValidFlow := FALSE;
END_METHOD

// 已中止狀態 — 等待 Reset 信號
METHOD M_STATE_ABORTED
VAR_INPUT
END_VAR
IF NOT _bRetry THEN
	Busy 	:= FALSE;
	Aborted := TRUE;
	Error 	:= TRUE;
	Status 	:= strStatus;
	_AbortCompleted := FALSE;
	uiAbortingStep  := 0;
END_IF
// 判斷內部Serivce 已經在aborted 狀態等著才能讓 FB reset
IF fbSingleFlow.eState = STATE_Aborted THEN
	IF reset THEN
		fbSingleFlow();
		fbSingleFlow.Reset := TRUE;

		_bRetry := TRUE;
		Aborted	:= FALSE;
		Error	:= FALSE;
	END_IF
END_IF

// 狀態機切換
IF NOT Execute THEN
	eState := STATE_RESETTING;
ELSIF Execute AND _bRetry THEN
	IF fbSingleFlow.eState = STATE_EXECUTING THEN
		fbSingleFlow.Reset := FALSE;
		IF uiResumeStep > 0 THEN
			status			:= '';
			uiExecutingStep := uiResumeStep;
			eState 			:= STATE_EXECUTING;
		END_IF
	END_IF
END_IF


//IF __ISVALIDREF(BatchInfo) THEN
//	IF BatchInfo.HandShake.Reset THEN
//		IF uiResumeStep > 0 THEN
//			uiExecutingStep := uiResumeStep;
//			_bRetry := TRUE;
//		END_IF
//		eState := STATE_RESETTING;
//	END_IF
//ELSIF Reset THEN
//	IF uiResumeStep > 0 THEN
//		uiExecutingStep := uiResumeStep;
//		_bRetry := TRUE;
//	END_IF
//	eState := STATE_RESETTING;
//END_IF
END_METHOD

// 中止狀態 — 先停止單筆 FB
METHOD M_STATE_ABORTING
VAR_INPUT
END_VAR
CASE uiAbortingStep OF
	0:
		_Abort  := FALSE;
		_bRetry := FALSE;
		tonTimeOut.IN := FALSE;
		IF _bSingleFlowStarted THEN
			fbSingleFlow.Abort := TRUE;
			fbSingleFlow();
		END_IF
		uiAbortingStep := 100;
	
	100:
		fbSingleFlow();
		IF fbSingleFlow.Aborted OR NOT fbSingleFlow.Busy THEN
			fbSingleFlow.Abort := FALSE;
			uiAbortingStep := 9999;
		END_IF
	
	9999:
		_AbortCompleted := TRUE;
END_CASE

IF NOT Execute THEN
	eState := STATE_RESETTING;
ELSIF Execute AND _AbortCompleted THEN
	eState := STATE_Aborted;
END_IF
END_METHOD

// 完成狀態 — 等待外部取消 Execute
METHOD M_STATE_DONE
VAR_INPUT
END_VAR
Busy   := FALSE;
_Error := Error := FALSE;
_Abort := Abort := FALSE;
Done   := TRUE;

IF __ISVALIDREF(BatchInfo) THEN
	IF NOT BatchInfo.HandShake.Execute THEN
		eState := STATE_RESETTING;
	END_IF
ELSIF NOT Execute THEN
	eState := STATE_RESETTING;
END_IF
END_METHOD

// 休眠狀態 — 清除旗標,監聽 BatchInfo.HandShake.Execute 觸發
METHOD M_STATE_DORMANT
VAR_INPUT
END_VAR
Busy				:= FALSE;
Done				:= FALSE;
Aborted				:= FALSE;
Error				:= FALSE;
ErrorID				:= 0;
Status				:= '';
_ResetCompleted		:= FALSE;
_Error				:= FALSE;
_Executed			:= FALSE;
_Abort				:= FALSE;
uiExecutingStep		:= 0;
uiResettingStep		:= 0;
uiResumeStep		:= 0;
uiAbortingStep		:= 0;

tonTimeOut.IN		:= FALSE;
_UniqueErrorCode	:= '0';

iProcessingIndex	:= 0;
_bSingleFlowStarted	:= FALSE;

IF __ISVALIDREF(BatchInfo) THEN
	MEMSET(ADR(BatchInfo.WorkedID), 0, SIZEOF(BatchInfo.WorkedID));
END_IF

_AbortCompleted		:= FALSE;
_bRetry				:= FALSE;

IF Execute THEN
	eState := STATE_EXECUTING;
END_IF

//IF __ISVALIDREF(BatchInfo) THEN
//	IF BatchInfo.HandShake.Execute AND NOT Stop THEN
//		Execute := TRUE;
//		eState := STATE_EXECUTING;
//	END_IF
//	IF BatchInfo.HandShake.Reset THEN
//		Reset := TRUE;
//	END_IF
//END_IF
END_METHOD

// 錯誤狀態 — 顯示錯誤訊息
METHOD M_STATE_ERROR
VAR_INPUT
END_VAR
Busy := FALSE;
Error := TRUE;
Status := strStatus;

IF NOT Execute THEN
	eState := STATE_RESETTING;
END_IF

//IF __ISVALIDREF(BatchInfo) THEN
//	IF NOT BatchInfo.HandShake.Execute THEN
//		eState := STATE_RESETTING;
//	END_IF
//ELSIF NOT Execute THEN
//	eState := STATE_RESETTING;
//END_IF
END_METHOD

// 執行主狀態 — 迭代批次中每筆有效流程
// 步序:
//   0:      M_FindNextValidFlow → 找到跳 100 / 沒找到跳 99000
//   100:    強制清 handshake + 配置 fbSingleFlow + 啟動 (HandshakeMode := TRUE)
//   200:    每 cycle 呼叫 fbSingleFlow, 等 Done 跳 300, 等 Error/Aborted abort
//   300:    寫 WorkedID + 強制清 ReadComplete + 釋放 fbSingleFlow
//   310:    等 fbSingleFlow 回 DORMANT, iProcessingIndex+1, 重置 timer 回 0
//   99000:  全部完成
METHOD M_STATE_EXECUTING
VAR_INPUT
END_VAR
Busy := TRUE;
tonTimeOut.IN := TRUE;

// 非自動模式直接中止
IF GVL_Machine.PackTags[UnitNo.Storage].Status.UnitModeCurrent <> E_UnitMode.Auto THEN
	strStatus := 'FB_FeedInRoundBeltBoxBatch: Not in Auto mode';
	_UniqueErrorCode := 'E_NOT_AUTO_MODE';
	_Abort := TRUE;
	RETURN;
END_IF

// Pause: 僅在迭代邊界 (step 0/310) 生效
IF __ISVALIDREF(BatchInfo) AND BatchInfo.Pause THEN
	IF uiExecutingStep = 0 OR uiExecutingStep = 310 THEN
		strStatus := 'FB_FeedInRoundBeltBoxBatch: Paused (at iteration boundary)';
		RETURN;
	END_IF
END_IF

// Per-iteration timeout (600s, step 310 推進時重置)
IF tonTimeOut.Q THEN
	strStatus := 'FB_FeedInRoundBeltBoxBatch: Batch per-iteration timeout';
	_UniqueErrorCode := 'E_BATCH_TIMEOUT';
	uiResumeStep := 100;
	_Abort := TRUE;
	RETURN;
END_IF

CASE uiExecutingStep OF

// ===== Step 0: 尋找下一筆有效流程 =====
0:
	IF NOT M_FindNextValidFlow() THEN
		uiExecutingStep := 99000;
	ELSE
		strStatus := CONCAT('Processing flow #', INT_TO_STRING(iProcessingIndex));
		uiExecutingStep := 100;
	END_IF

// ===== Step 100: 配置並啟動單筆 FB =====
100:
	// Safety: 強制清 handshake 確保 C# 看到本迭代 FeedBack 上升緣
	IF __ISVALIDREF(BatchInfo) THEN
		BatchInfo.FeedBack := FALSE;
		BatchInfo.ReadComplete := FALSE;
	END_IF
	fbSingleFlow.ReadComplete := FALSE;

	// 配置參照與 input
	fbSingleFlow.Robot REF= Robot;
	fbSingleFlow.RoundBelt REF= RoundBelt;
	fbSingleFlow.WareHouse REF= WareHouse;
	fbSingleFlow.Input := Input;
	fbSingleFlow.Info.ClampA_Setting := CurrentFlow.ClampA_Setting;
	fbSingleFlow.Info.ClampB_Setting := CurrentFlow.ClampB_Setting;
	fbSingleFlow.Stop := Stop;
	fbSingleFlow.HandshakeMode := TRUE;	// 啟用 ActionRecord + FeedBack/ReadComplete
	fbSingleFlow.Execute := TRUE;
	_bSingleFlowStarted := TRUE;
	uiExecutingStep := 200;

// ===== Step 200: 等待單筆 FB 完成 =====
200:
	fbSingleFlow();
	IF fbSingleFlow.Done THEN
		uiExecutingStep := 300;
	ELSIF fbSingleFlow.Error OR fbSingleFlow.Aborted THEN
		strStatus := CONCAT('Flow #', CONCAT(INT_TO_STRING(iProcessingIndex), ' failed'));
		_UniqueErrorCode := 'E_FLOW_FAILED';
		uiResumeStep := 100;	// retry 從重配置開始
		_Abort := TRUE;
	END_IF

// ===== Step 300: 記錄完成 + 釋放單筆 FB =====
300:
	IF __ISVALIDREF(BatchInfo) THEN
		BatchInfo.WorkedID[iProcessingIndex] := CurrentFlow.ID;
		BatchInfo.ReadComplete := FALSE;	// Safety: 防 C# 殘留
	END_IF
	fbSingleFlow.Execute := FALSE;
	fbSingleFlow();
	_bSingleFlowStarted := FALSE;
	uiExecutingStep := 310;

// ===== Step 310: 等 fbSingleFlow 回 DORMANT 後再推進 =====
310:
	fbSingleFlow();
	IF NOT fbSingleFlow.Busy AND NOT fbSingleFlow.Done AND NOT fbSingleFlow.Error THEN
		iProcessingIndex := iProcessingIndex + 1;
		tonTimeOut.IN := FALSE;	// per-iteration timer 重置
		uiExecutingStep := 0;
	END_IF

// ===== Step 99000: 全部完成 =====
99000:
	_Executed := TRUE;

END_CASE

// ===== 狀態切換 =====
IF NOT Execute THEN
	eState := STATE_RESETTING;
ELSIF _Error THEN
	eState := STATE_ERROR;
ELSIF _Abort THEN
	eState := STATE_ABORTING;
ELSIF _Executed THEN
	eState := STATE_DONE;
END_IF
END_METHOD

// 重置狀態 — 等待 fbSingleFlow 回 DORMANT 後決定走 retry 或正常路徑
METHOD M_STATE_RESETTING
VAR_INPUT
END_VAR
// Done := false 更改到Dormant 清除確保，上位檢查到done 後可以直接下Execute

CASE uiResettingStep OF
	0:
		Error := FALSE;
		Aborted := FALSE;
		tonTimeOut.IN := FALSE;

		fbSingleFlow();
		fbSingleFlow.Execute := FALSE;
		uiResettingStep := 50;

	50:
//		// 每 scan call fbSingleFlow 推進其內部 RESETTING → DORMANT
//		// (移除 A00 的 freerun call 後,這裡是 RESETTING 期間唯一的驅動點)
//		fbSingleFlow();
//		IF fbSingleFlow.eState = STATE_DORMANT THEN
//			IF _bRetry THEN
//				_bRetry := FALSE;
//				eState := STATE_EXECUTING;
//				RETURN;
//			END_IF
//			uiResettingStep := 100;
//		END_IF
		IF fbSingleFlow.eState = STATE_DORMANT THEN
			uiResettingStep := 100;
		END_IF

	100:
//		Done := FALSE;
//		Busy := FALSE;
		_ResetCompleted := TRUE;

END_CASE

IF _ResetCompleted THEN
	eState := STATE_DORMANT;
END_IF
END_METHOD

END_FUNCTION_BLOCK

// ---- Library/20_MachineUnits/21_StorageArea/Service_Robot/FB_RobotSelfHoming.TcPOU
FUNCTION_BLOCK FB_RobotSelfHoming EXTENDS FB_ObjectBase_V2 IMPLEMENTS IBasicElement
VAR_INPUT
	FanucRobot		: REFERENCE TO FB_FanucRobot_Basic_V2;
	Input			: REFERENCE TO ST_InputTable;
	Output			: REFERENCE TO ST_OutputTable;
	Motor			: REFERENCE TO UNI_MotorList;
	
	
	BypassFeedOutToNGCV	: BOOL;
END_VAR
VAR_OUTPUT
END_VAR
VAR
	binjectVelPara	 : BOOL;
	_RobotFeedOutVel : UINT :=20  ;
	RobotRunningVel	 : UINT;
	
	// Reboot Timer
	TON_RobotRebootDelay		: TON;		// 手臂電源復位延遲
	TON_RobotRebootTimeOut		: TON;		// 手臂重啟斷訊回歸延遲
	TON_RobotErrorDetectDelay	: TON;		// 手臂偵測錯誤延遲
	TON_ServiceTimeOut			: TON;		
	
	//Internal Robot FeedOut To NGCV use
	TON_RobotFeedOutCommand : TON;			// 手臂放盒至 NG軌道 Command 計時
	TON_RobotTimeOut		: TON;			// 手臂放盒至 NG軌道 Service done 計時
	
	_fbRobotRegionMove_FeedInConveyor :  FB_RobotRegionMove_FeedInConveyor_V2;
END_VAR

SUPER^.A10_StateControl();
A00_BasicUnits();

ACTION A00_BasicUnits:
TON_RobotRebootDelay(		PT := T#2S);
TON_RobotRebootTimeOut(		PT := T#60S);
TON_RobotErrorDetectDelay(	PT := T#3S);
TON_ServiceTimeOut(			PT := T#120S);
TON_RobotFeedOutCommand(	PT:= T#5S);
TON_RobotTimeOut(			PT := T#60S);

_fbRobotRegionMove_FeedInConveyor(
	Execute:= , 
	Abort:= , 
	Reset:= , 
	ObjectName:= , 
	Busy=> , 
	Done=> , 
	Aborted=> , 
	Error=> , 
	ErrorID=> , 
	Status=> , 
	UniqueErrorCode=> , 
	Robot:= FanucRobot, 
	LowerConveyor:= Motor.List.LowCV, 
	Input:= input, 
	Info:= , 
	Stop:= );
END_ACTION

METHOD M_CheckCommand : BOOL
VAR_INPUT
END_VAR
IF GVL_ADS.AutoMode_RobotAbsMove.HandShake.Execute 
	OR GVL_ADS.AutoMode_FeedInEmptyBoxWithRobot.Command.Execute 
	OR GVL_ADS.AutoMode_FeedInRoundBeltBoxToWareHouse.Command.Execute
	OR GVL_ADS.AutoMode_ReloadRoundBeltBoxWithRobot.Command.Execute 
	OR GVL_ADS.AutoMode_RobotRegionMove_AllocatedConveyor.Command.Execute
	OR GVL_ADS.AutoMode_RobotRegionMove_BufferArea.Command.Execute
	OR GVL_ADS.AutoMode_RobotRegionMove_FeedInConveyor.Command.Execute
	OR GVL_ADS.AutoMode_RobotRegionMove_PullOutConveyor.Command.Execute
	OR GVL_ADS.AutoMode_RobotRegionMove_RoundBelt.Command.Execute
	OR GVL_ADS.AutoMode_WarehouseMotoWithRobotMove.HandShake.Execute 
THEN
	M_CheckCommand := FALSE;
ELSE
	M_CheckCommand := TRUE;
END_IF
END_METHOD

METHOD  M_STATE_ABORTED
VAR_INPUT
END_VAR

Busy  := FALSE;
Error := TRUE;
Aborted := TRUE;
uiAbortingStep 	:= 0;
_AbortCompleted := FALSE;

// 狀態機切換
IF NOT Execute THEN
	eState := STATE_RESETTING;
ELSIF Execute AND reset THEN
	Error	:= false;
	Aborted	:= false;
	eState 	:= STATE_EXECUTING;
END_IF
END_METHOD

METHOD  M_STATE_ABORTING
VAR_INPUT
END_VAR

CASE uiAbortingStep OF
	0 :
		_Abort := FALSE;
		TON_RobotRebootDelay.IN 	:= FALSE;
		TON_RobotRebootTimeOut.IN	:= FALSE;
		TON_RobotErrorDetectDelay.IN:= FALSE;
		TON_ServiceTimeOut.IN		:= FALSE;
		TON_RobotFeedOutCommand.IN	:= FALSE;
		TON_RobotTimeOut.IN			:= FALSE;
		
		uiAbortingStep:=9999;

	9999:	
		_AbortCompleted:=TRUE;
END_CASE

IF _AbortCompleted THEN	
	eSTATE :=STATE_ABORTED;
END_IF
END_METHOD

METHOD  M_STATE_DONE
VAR_INPUT
END_VAR
Busy   := FALSE;
_Error := Error := FALSE;
_Abort := Abort := FALSE;
Done   := TRUE;

IF NOT Execute THEN
    eState := STATE_RESETTING;
END_IF
END_METHOD

METHOD  M_STATE_DORMANT
VAR_INPUT
END_VAR

Busy 			:= FALSE;
Done 			:= FALSE;
Aborted 		:= FALSE;
Error			:= FALSE;
Paused			:= FALSE;
ErrorID			:= 0;
Status			:= '';
UniqueErrorCode := '';

_Executed 			:= FALSE;
_Error				:= FALSE;
_Abort				:= FALSE;
_ResetCompleted 	:= FALSE;
_AbortCompleted 	:= FALSE;
_HoldingCompleted 	:= FALSE;
_HeldCompleted	 	:= FALSE;
_UnholdCompleted 	:= FALSE;

uiExecutingStep 		:= 0;
uiResettingStep 		:= 0;
uiAbortingStep 			:= 0;
uiHoldingStep			:= 0;
uiHeldStep				:= 0;
uiUnholdStep			:= 0;

TON_RobotRebootDelay.IN 	:= FALSE;
TON_RobotRebootTimeOut.IN	:= FALSE;
TON_RobotErrorDetectDelay.IN:= FALSE;
TON_ServiceTimeOut.IN		:= FALSE;
TON_RobotFeedOutCommand.IN	:= FALSE;
TON_RobotTimeOut.IN			:= FALSE;

IF Execute THEN
    eState := STATE_EXECUTING;
END_IF
END_METHOD

METHOD  M_STATE_ERROR
VAR_INPUT
END_VAR

ERROR   := TRUE;
Busy	:= FALSE;
_Error	:= false;

IF NOT Execute THEN	
	Error	:= FALSE;
	eSTATE	:=STATE_RESETTING;
END_IF
END_METHOD

METHOD  M_STATE_EXECUTING
VAR_INPUT
END_VAR
busy := true;

// 暫停
IF Pause THEN 
	_HoldingCompleted 	:= FALSE;
	_HeldCompleted	 	:= FALSE;
	_UnholdCompleted 	:= FALSE;
	uiHoldingStep		:= 0;
	uiHeldStep			:= 0;
	uiUnholdStep		:= 0;
	eState    			:= STATE_Holding;
END_IF
IF TON_ServiceTimeOut.Q THEN
	status	:= 'FB_RobotSelfHoming: Service TimeOut';
	_Error	:= TRUE;
END_IF
IF GVL_HMI.Setup.StorageRobot.RobotVelocity = 0 THEN
	_Error := TRUE;
	status := 'FB_RobotSelfHoming: Robot Speed cannot be 0 ';
	eState := STATE_ERROR;
	RETURN;
END_IF

// 動作主流程 狀態機
CASE uiExecutingStep OF
	
	0:		
			IF GVL_Machine.PackTags[UnitNo.Storage].Status.UnitModeCurrent <> E_UnitMode.Auto THEN
				Status := 'FB_RobotSelfHoming Step 0: Not in Auto mode';
				_Error := TRUE;
			ELSE
				uiExecutingStep := 50;
			END_IF

	50:		// 檢查是否有其他的手臂程式正在執行。
			TON_ServiceTimeOut.IN := TRUE;
			IF NOT binjectVelPara THEN
				binjectVelPara	:= TRUE;
				RobotRunningVel := LREAL_TO_UINT( GVL_HMI.Setup.StorageRobot.RobotVelocity);
			END_IF
			
			IF M_CheckCommand() THEN
				uiExecutingStep := 100;
			ELSE
				status := 'FB_RobotSelfHoming Step 50: Wrong Command : another Robot Service Executing';
				_Error := TRUE;
			END_IF
	
	100:
			IF FanucRobot._EIPConnectionState = 8195 THEN
				Output.bStorage_FanucRobotPower := TRUE;
				TON_RobotRebootDelay.IN 		:= TRUE;
				TON_RobotRebootTimeOut.IN		:= TRUE;
			ELSE
				uiExecutingStep := 200;
			END_IF
			IF TON_RobotRebootDelay.Q THEN
				output.bStorage_FanucRobotPower := FALSE;
			END_IF
			IF TON_RobotRebootTimeOut.Q THEN
				status := 'FB_RobotSelfHoming Step 100: Robot Reboot Timeout';
				_Error := TRUE;
			END_IF
			
	200:	// Robot 斷訊恢復後重新下回 home 命令
			TON_RobotRebootDelay.IN			:= FALSE;
			TON_RobotRebootTimeOut.IN		:= FALSE;
			FanucRobot.OpMode := E_FanucRobotOpMode.RSR02;		//Restart Robot Homing
			TON_RobotErrorDetectDelay.IN := TRUE;
			IF TON_RobotErrorDetectDelay.Q THEN
				uiExecutingStep := 500;
			END_IF
	500:
			IF FanucRobot._RSR2_Completed THEN
				uiExecutingStep := 600;
			END_IF
			
	600:
			FanucRobot.OpMode := E_FanucRobotOpMode.RSR01;
			IF FanucRobot._RSR1_Ready THEN
				uiExecutingStep := 700;
			END_IF
	700:
			IF FanucRobot.OpMode = E_FanucRobotOpMode.RSR01 AND NOT FanucRobot._DI1.Done AND FanucRobot._DI12.RSR1_Active THEN
				uiExecutingStep := 1050;
			END_IF
	1050:
			IF BypassFeedOutToNGCV THEN
				uiExecutingStep := 9999;
			ELSE
				uiExecutingStep := 1100;
			END_IF
			
	1100:	//detect Robot Clamp ,, if clamp have box or clamp not open todo 
			IF NOT FanucRobot._DI1.ClampA_Open AND NOT FanucRobot._DI1.ClampB_Open  THEN
				GVL_HMI.Setup.StorageRobot.RobotVelocity := _RobotFeedOutVel;
				uiExecutingStep := 2000;
			ELSIF NOT FanucRobot._DI1.ClampA_Open  THEN
				GVL_HMI.Setup.StorageRobot.RobotVelocity := _RobotFeedOutVel;
				uiExecutingStep := 3000;
			ELSIF NOT FanucRobot._DI1.ClampB_Open  THEN
				GVL_HMI.Setup.StorageRobot.RobotVelocity := _RobotFeedOutVel;
				uiExecutingStep := 4000;
			ELSE 
				GVL_HMI.Setup.StorageRobot.RobotVelocity := RobotRunningVel;
				uiExecutingStep := 9999;
			END_IF
		
	2000:	// Both Clamp , not open and sensor detect
			TON_RobotFeedOutCommand.IN := TRUE;
			_fbRobotRegionMove_FeedInConveyor.M_StartHomingFeedOut(UseA := TRUE,
												UseB := TRUE);
			IF _fbRobotRegionMove_FeedInConveyor.Busy THEN
				uiExecutingStep := 2100;
			END_IF
			IF TON_RobotFeedOutCommand.Q THEN
				status := 'FB_RobotSelfHoming Step 2000: Storage FanucRobot FeedOut TO NG Conveyor NOT busy';
				_Error := TRUE;
			END_IF

	2100:	// FeedOut done clear command
			TON_RobotFeedOutCommand.IN  := FALSE;		//check command
			TON_RobotTimeOut.IN 		:= TRUE;		//Robot FeeOut Timer
			IF _fbRobotRegionMove_FeedInConveyor.Done THEN
				_fbRobotRegionMove_FeedInConveyor.M_ResetHomingFeedOut();
				uiExecutingStep := 0;
			END_IF
			IF TON_RobotTimeOut.Q THEN
				status := 'FB_RobotSelfHoming Step 2100: Storage FanucRobot FeedOut to NG Conveyor Done Timeout';
				_Error := TRUE;
			END_IF
		
	3000:	//Clamp A
			TON_RobotFeedOutCommand.IN := TRUE;
			_fbRobotRegionMove_FeedInConveyor.M_StartHomingFeedOut(UseA := TRUE,
												useB := FALSE);
			IF _fbRobotRegionMove_FeedInConveyor.Busy THEN
				uiExecutingStep := 3100;
			END_IF
			IF TON_RobotFeedOutCommand.Q THEN
				status := 'FB_RobotSelfHoming Step 3000: Storage FanucRobot FeedOut TO NG Conveyor NOT busy';
				_Error := TRUE;
			END_IF

	3100:	//FeedOut Done clear command
			TON_RobotFeedOutCommand.IN  := FALSE;		//check command
			TON_RobotTimeOut.IN 		:= TRUE;		//Robot FeeOut Timer
			IF _fbRobotRegionMove_FeedInConveyor.Done THEN
				_fbRobotRegionMove_FeedInConveyor.M_ResetHomingFeedOut();
				uiExecutingStep := 0;
			END_IF
			IF TON_RobotTimeOut.Q THEN
				status := 'FB_RobotSelfHoming Step 3100: Storage FanucRobot FeedOut to NG Conveyor Done Timeout';
				_Error := TRUE;
			END_IF

	4000:	//Clamp B
			TON_RobotFeedOutCommand.IN := TRUE;
			_fbRobotRegionMove_FeedInConveyor.M_StartHomingFeedOut(UseA := FALSE,
												useB := TRUE);
			IF _fbRobotRegionMove_FeedInConveyor.Busy THEN
				uiExecutingStep := 4100;
			END_IF
			IF TON_RobotFeedOutCommand.Q THEN
				status := 'FB_RobotSelfHoming Step 4000: Storage FanucRobot FeedOut TO NG Conveyor NOT busy';
				_Error := TRUE;
			END_IF

	4100:	//FeedOut Done clear command
			TON_RobotFeedOutCommand.IN  := FALSE;		//check command
			TON_RobotTimeOut.IN 		:= TRUE;		//Robot FeeOut Timer
			IF _fbRobotRegionMove_FeedInConveyor.Done THEN
				_fbRobotRegionMove_FeedInConveyor.M_ResetHomingFeedOut();
				uiExecutingStep := 0;
			END_IF
			IF TON_RobotTimeOut.Q THEN
				status := 'FB_RobotSelfHoming Step 4100: Storage FanucRobot FeedOut to NG Conveyor Done Timeout';
				_Error := TRUE;
			END_IF
			
	9999:
			status		:= 'FB_RobotSelfHoming Step 9999: Process done';
			_Executed 	:= TRUE;		
end_case

// 狀態機切換
IF NOT Execute THEN
	eState := STATE_RESETTING;
ELSIF _Error THEN
	eState := STATE_ERROR;
ELSIF _Abort THEN
	eState := STATE_ABORTING;
ELSIF _Executed THEN
	eState := STATE_DONE;
END_IF
END_METHOD

METHOD M_STATE_HELD
VAR_INPUT
END_VAR

Busy 	:= FALSE;
Paused 	:= TRUE;

CASE uiHeldStep OF
	0:
		uiHeldStep := 9999;

	9999:
		_HeldCompleted := TRUE;	

END_CASE

IF _HeldCompleted AND NOT Pause THEN
	eState := STATE_UnHold;
END_IF
END_METHOD

METHOD M_STATE_HOLDING
VAR_INPUT
END_VAR

CASE uiHoldingStep OF 
	0:	    // 需關閉 Timer 等等須暫停的變數
	
		TON_RobotRebootDelay.IN 	:= FALSE;
		TON_RobotRebootTimeOut.IN	:= FALSE;
		TON_RobotErrorDetectDelay.IN:= FALSE;
		TON_ServiceTimeOut.IN		:= FALSE;
		TON_RobotFeedOutCommand.IN	:= FALSE;
		TON_RobotTimeOut.IN			:= FALSE;
		
		uiHoldingStep := 9999;
		
	9999:	// holding 完成
		_HoldingCompleted := TRUE;
END_CASE

IF _HoldingCompleted THEN
	eState := STATE_Held;
END_IF
END_METHOD

METHOD  M_STATE_RESETTING
VAR_INPUT
END_VAR
// Done := false 更改到Dormant 清除確保，上位檢查到done 後可以直接下Execute

CASE uiResettingStep OF

	0:
			TON_RobotRebootDelay.IN 	:= FALSE;
			TON_RobotRebootTimeOut.IN	:= FALSE;
			TON_RobotErrorDetectDelay.IN:= FALSE;
			TON_ServiceTimeOut.IN		:= FALSE;
			TON_RobotFeedOutCommand.IN	:= FALSE;
			TON_RobotTimeOut.IN			:= FALSE;

			_fbRobotRegionMove_FeedInConveyor.M_ResetHomingFeedOut();

			uiResettingStep := 9999;
	9999:
//			Done := FALSE;
//			Busy := FALSE;
			_ResetCompleted:=TRUE;
END_CASE

IF _ResetCompleted THEN
	eSTATE:=STATE_DORMANT;
END_IF
END_METHOD

METHOD M_STATE_UNHOLD
VAR_INPUT
END_VAR

CASE uiUnholdStep OF 
	0:		
		uiUnholdStep := 9999;
		
	9999:
		_UnholdCompleted := TRUE;
		
END_CASE

IF _UnholdCompleted THEN
	Paused := FALSE;
	eState := STATE_EXECUTING;
END_IF
END_METHOD

END_FUNCTION_BLOCK

// ---- Library/20_MachineUnits/21_StorageArea/Service/FB_StorageHoming.TcPOU
FUNCTION_BLOCK FB_StorageHoming EXTENDS FB_ActionBasic
VAR_INPUT
	xExecute 	: BOOL;
	xAbort 		: BOOL;
    Cylinder    : REFERENCE TO UNI_CylinderList;
    Motor       : REFERENCE TO UNI_MotorList;
    FanucRobot  : REFERENCE TO FB_FanucRobot_Basic_V2;
	Homed 		: REFERENCE TO BOOL;
	Output		: REFERENCE TO ST_OutputTable;
	Input		: REFERENCE TO ST_InputTable;
	Service		: REFERENCE TO ST_StorageService;
END_VAR
VAR_OUTPUT
	xAborted : BOOL;
	iErrorID : INT;
	ErrorMsg : STRING;
	RobotResetCMD : BOOL;
	RackMotorHomeRequest : BOOL;
END_VAR
VAR
	StateBehaviour 		: CBML.ETrigA;
	uiStorageHomingStep : UINT;
	CylinderCheckTon 	: TON;
	MotorCheckTon 		: TON;
	FanucRobotCheckTon  : TON;
	ResetRobotDelay	 	: TON;
	TON_RobotFeedOutCommand : TON;
	TON_RobotTimeOut		: TON;
	fbExecuteEdgeDetect :FB_EdgeDetect;
	_fbRobotRegionMove_FeedInConveyor :  FB_RobotRegionMove_FeedInConveyor_V2;
	
		// EIP 斷線恢復用計時器
	tonPowerCycle			: TON;		// 電源 TRUE 維持 5 秒
	tonPowerCycleTimeout	: TON;		// 電源 FALSE 後等待重連 60 秒

	// 啟動延時 - 等待心跳偵測完成 (冷啟動用)
	tonStartupDelay			: TON;		// 啟動延時 5 秒

END_VAR

THIS^.IBehaviourModel := StateBehaviour;
A00_BasicUnits();
StateBehaviour(xExecute := xExecute,
    xDone => xDone,
    xBusy => xBusy,
    xError => xError,
    xAbort := xAbort OR fbExecuteEdgeDetect.xFallingEdge,
    xAborted => xAborted);

//Error Msg
iErrorID := StateBehaviour._model.iErrorID;
ErrorMsg := M_GetErrorMsg(xErrorID := iErrorID);

//Make sure that C# turns off execute to shut down the service
fbExecuteEdgeDetect(xInput :=xExecute);

ACTION A00_BasicUnits:
CylinderCheckTon(PT := T#5S);
MotorCheckTon(PT := T#2S);
FanucRobotCheckTon(PT:=T#120S);
ResetRobotDelay(PT:=T#300MS);
TON_RobotFeedOutCommand(PT:= T#5S);
TON_RobotTimeOut(PT := T#60S);
tonPowerCycle(PT := T#5S);			// 電源維持 TRUE 5 秒
tonPowerCycleTimeout(PT := T#60S);	// 電源 FALSE 後等待重連 60 秒
tonStartupDelay(PT := T#5S);		// 啟動延時 5 秒 (等待心跳偵測)


_fbRobotRegionMove_FeedInConveyor(
	Execute:= , 
	Abort:= , 
	Reset:= , 
	ObjectName:= , 
	Busy=> , 
	Done=> , 
	Aborted=> , 
	Error=> , 
	ErrorID=> , 
	Status=> , 
	UniqueErrorCode=> , 
	Robot:= FanucRobot, 
	LowerConveyor:= Motor.List.LowCV, 
	Input:= input, 
	Info:= , 
	Stop:= );
END_ACTION

METHOD CleanupAction
VAR_INPUT
    xAbortProposed : BOOL;
    iErrorIDProposed: INT;
END_VAR
VAR_OUTPUT
    xComplete : BOOL := TRUE;
    xAbort: BOOL := xAbortProposed;
 	iErrorID : INT := iErrorIDProposed;
END_VAR
END_METHOD

METHOD CyclicAction
VAR_INPUT
    itfTimingController : CBML.ITimingController;
END_VAR
VAR_OUTPUT
    xComplete : BOOL := TRUE;
    iErrorID : INT := 0;
END_VAR
VAR
	tehn: INT;
END_VAR
xComplete := FALSE;
CASE uiStorageHomingStep OF
	0: // Retract Cylinder
		TON_RobotFeedOutCommand.IN  := FALSE;
		TON_RobotTimeOut.IN 		:= FALSE;
		M_RetractStorageCylinder();
		RobotResetCMD := FALSE;	
		Cylinder.List.fbStackPush.M_Retract();
		IF Cylinder.List.fbStackPush.InRearPosition THEN		// safecheck Rackmotor home 
		uiStorageHomingStep := 100;
		END_IF
	100:
		IF M_CheckStorageCylinderInRear() THEN
			uiStorageHomingStep := 200;
		ELSE
			CylinderCheckTon.IN := TRUE;
			IF CylinderCheckTon.Q THEN
				iErrorID := 2;
			END_IF
		END_IF
	200:
			CylinderCheckTon.IN := FALSE;
			M_StopStorageMotor ();
			uiStorageHomingStep := 300;
	300:
		IF M_CheckStorageMotorInStop() THEN
			uiStorageHomingStep := 390;
		ELSE
			MotorCheckTon.IN := TRUE;
			IF MotorCheckTon.Q THEN
				iErrorID := 3;
			END_IF
		END_IF
	// ============================================================================
	// Step 390: 啟動延時 - 等待心跳偵測完成
	// - 冷啟動時，心跳偵測需要 5 秒 (10 × 0.5s) 才能判定連線狀態
	// - 必須等心跳偵測完成後，才能正確判斷機器人是否已連線
	// ============================================================================
	390:
		MotorCheckTon.IN := FALSE;
		FanucRobotCheckTon.IN := TRUE;
		RobotResetCMD := FALSE;
		tonStartupDelay.IN := TRUE;

		// 等待 5 秒讓心跳偵測完成
		IF tonStartupDelay.Q THEN
			tonStartupDelay.IN := FALSE;
			uiStorageHomingStep := 400;
		END_IF

	// ============================================================================
	// Step 400: 檢查機器人連線狀態
	// - 心跳偵測已完成，現在可以正確判斷連線狀態
	// ============================================================================
	400:
		// 斷線判定: EIP scanner 報斷線 OR 軟體心跳 5 秒未翻轉 (iTestCnt >= 10)
		IF FanucRobot._EIPConnectionState = 8195 OR FanucRobot.iTestCnt >= 10 THEN
			// EIP/心跳 斷線，執行電源循環恢復
			uiStorageHomingStep := 440;
		ELSIF FanucRobot.Halt THEN
			// Robot 在 Halt 狀態 → 清除 Hold 讓 Halt 解除，再 Reset 回 DORMANT
			FanucRobot.Hold := FALSE;
			FanucRobot.Reset := TRUE;
			ResetRobotDelay.IN := TRUE;
		ELSIF FanucRobot.Error THEN
			// 一般錯誤，執行正常重置
			RobotResetCMD := TRUE;
			ResetRobotDelay.IN := TRUE;
		ELSIF FanucRobot._UO1.UO03_PrgRunning THEN
			// Robot 正在執行流程 → 強制停止後再切 RSR02
			FanucRobot.M_ResetAllCommand();
			FanucRobot.Hold := FALSE;
			FanucRobot.Reset := TRUE;
			ResetRobotDelay.IN := TRUE;
		ELSE
			uiStorageHomingStep := 500;
		END_IF
		IF ResetRobotDelay.Q THEN
			ResetRobotDelay.IN := FALSE;
			FanucRobot.Reset := FALSE;
			uiStorageHomingStep := 500;
		END_IF

	440:	// EIP 斷線恢復: 電源 TRUE
		RobotResetCMD := FALSE;
		ResetRobotDelay.IN := FALSE;
		FanucRobotCheckTon.IN := FALSE;					// 暫停 120 秒總超時，避免電源循環中誤觸發
		OutPut.bStorage_FanucRobotPower := TRUE;		// 強制電源 TRUE
		tonPowerCycle.IN := TRUE;						// 開始 5 秒計時
		tonPowerCycleTimeout.IN := FALSE;				// 還不開始重連計時
		uiStorageHomingStep := 450;

	450:	// EIP 斷線恢復: 等待 5 秒
		IF tonPowerCycle.Q THEN
			// 5 秒到，電源 FALSE，開始計時等待重連
			tonPowerCycle.IN := FALSE;
			OutPut.bStorage_FanucRobotPower := FALSE;
			tonPowerCycleTimeout.IN := TRUE;			// 現在開始 60 秒重連計時
			uiStorageHomingStep := 460;
		END_IF

	460:	// EIP 斷線恢復: 等待重新連線 (60秒超時)
		IF tonPowerCycleTimeout.Q THEN
			// 超時 60 秒，報錯
			tonPowerCycleTimeout.IN := FALSE;
			iErrorID := 22;
			uiStorageHomingStep := 9999;
		ELSIF FanucRobot._EIPConnectionState <> 8195 AND FanucRobot.iTestCnt < 10 THEN
			// EIP 已重連 + 心跳已恢復，繼續執行 RSR02
			tonPowerCycleTimeout.IN := FALSE;
			FanucRobotCheckTon.IN := TRUE;				// 恢復 120 秒總超時監控
			uiStorageHomingStep := 500;
		END_IF

	500:
		RobotResetCMD := FALSE;
		RackMotorHomeRequest := TRUE;		//RackMotor Homing	edit by min 20250716
		FanucRobot.OpMode := E_FanucRobotOpMode.RSR02;
		// RSR02 執行中不檢查錯誤，讓 RSR02 完成後再檢查
		IF FanucRobot._RSR2_Completed THEN
			uiStorageHomingStep := 600;
		END_IF
	600:
		FanucRobot.OpMode := E_FanucRobotOpMode.RSR01;
		IF FanucRobot._RSR1_Ready AND
			arAxisCtrl_gb[AxisNo.RackMotor].Admin.Axis.Status.Homed
		THEN
			uiStorageHomingStep := 1000;
		END_IF
			// RSR02 完成後，檢查是否還有錯誤
		IF FanucRobot.Error THEN
			iErrorID := 21;		// RSR02 完成但錯誤仍存在
		END_IF
	1000:	
			IF FanucRobot.OpMode = E_FanucRobotOpMode.RSR01 AND NOT FanucRobot._DI1.Done AND FanucRobot._DI12.RSR1_Active THEN
				uiStorageHomingStep := 1100;
				//uiStorageHomingStep := 9000;
			END_IF
			
	1100:	//detect Robot Clamp ,, if clamp have box or clamp not open todo 
			IF NOT FanucRobot._DI1.ClampA_Open AND NOT FanucRobot._DI1.ClampB_Open  THEN
				uiStorageHomingStep := 2000;
			ELSIF NOT FanucRobot._DI1.ClampA_Open  THEN
				uiStorageHomingStep := 3000;
			ELSIF NOT FanucRobot._DI1.ClampB_Open  THEN
				uiStorageHomingStep := 4000;
			ELSE 
				uiStorageHomingStep := 9000;
			END_IF
		
	2000:	// Both Clamp , not open and sensor detect
			TON_RobotFeedOutCommand.IN := TRUE;
			_fbRobotRegionMove_FeedInConveyor.M_StartHomingFeedOut(UseA := TRUE,
												UseB := TRUE);
			IF _fbRobotRegionMove_FeedInConveyor.Busy THEN
				uiStorageHomingStep := 2100;
			END_IF
			IF TON_RobotFeedOutCommand.Q THEN
				iErrorID := 10;
			END_IF
		
	2100:	// FeedOut done clear command 
			TON_RobotFeedOutCommand.IN  := FALSE;		//check command 
			TON_RobotTimeOut.IN 		:= TRUE;		//Robot FeeOut Timer
			IF _fbRobotRegionMove_FeedInConveyor.Done THEN
				_fbRobotRegionMove_FeedInConveyor.M_ResetHomingFeedOut();
				uiStorageHomingStep := 0;
			END_IF
			IF TON_RobotTimeOut.Q THEN
				iErrorID := 11;
			END_IF
		
	3000:	//Clamp A 
			TON_RobotFeedOutCommand.IN := TRUE;
			_fbRobotRegionMove_FeedInConveyor.M_StartHomingFeedOut(UseA := TRUE,
												useB := FALSE);
			IF _fbRobotRegionMove_FeedInConveyor.Busy THEN
				uiStorageHomingStep := 3100;
			END_IF
			IF TON_RobotFeedOutCommand.Q THEN
				iErrorID := 10;
			END_IF
		
	3100:	//FeedOut Done clear command
			TON_RobotFeedOutCommand.IN  := FALSE;		//check command 
			TON_RobotTimeOut.IN 		:= TRUE;		//Robot FeeOut Timer
			IF _fbRobotRegionMove_FeedInConveyor.Done THEN
				_fbRobotRegionMove_FeedInConveyor.M_ResetHomingFeedOut();
				uiStorageHomingStep := 0;
			END_IF
			IF TON_RobotTimeOut.Q THEN
				iErrorID := 11;
			END_IF
		
	4000:	//Clamp B
			TON_RobotFeedOutCommand.IN := TRUE;
			_fbRobotRegionMove_FeedInConveyor.M_StartHomingFeedOut(UseA := FALSE,
												useB := TRUE);
			IF _fbRobotRegionMove_FeedInConveyor.Busy THEN
				uiStorageHomingStep := 4100;
			END_IF
			IF TON_RobotFeedOutCommand.Q THEN
				iErrorID := 10;
			END_IF
		
	4100:	//FeedOut Done clear command
			TON_RobotFeedOutCommand.IN  := FALSE;		//check command 
			TON_RobotTimeOut.IN 		:= TRUE;		//Robot FeeOut Timer
			IF _fbRobotRegionMove_FeedInConveyor.Done THEN
				_fbRobotRegionMove_FeedInConveyor.M_ResetHomingFeedOut();
				uiStorageHomingStep := 0;
			END_IF
			IF TON_RobotTimeOut.Q THEN
				iErrorID := 11;
			END_IF
	9000:
		FanucRobotCheckTon.IN := FALSE;
		Homed := TRUE;
		xComplete := TRUE;
END_CASE

IF FanucRobotCheckTon.Q THEN
	iErrorID := 4;
END_IF
END_METHOD

METHOD ExitAction
VAR_INPUT
    xAfterCleanup : BOOL;
    xInCopyCode : BOOL;
END_VAR
uiStorageHomingStep := 0;
END_METHOD

METHOD M_CheckStorageCylinderInRear : BOOL
VAR_INPUT
END_VAR
M_CheckStorageCylinderInRear := Cylinder.List.fbUpCV_FeedInPress1.InRearPosition AND
    Cylinder.List.fbUpCV_FeedInPress2.InRearPosition AND
    Cylinder.List.fbUpCV_DiameterPress.InRearPosition AND
    Cylinder.List.fbUpCV_CamaraPress1.InRearPosition AND
    Cylinder.List.fbUpCV_CamaraPress2.InRearPosition AND
    Cylinder.List.fbUpCV_CamaraPress3.InRearPosition AND
    Cylinder.List.fbUpCV_CamaraPress4.InRearPosition AND
    Cylinder.List.fbUpCV_Block1.InRearPosition AND
    Cylinder.List.fbUpCV_Block2.InRearPosition AND
    Cylinder.List.fbUpCV_Block3.InRearPosition AND
    Cylinder.List.fbUpCV_DiameterHoriz.InRearPosition AND
    Cylinder.List.fbUpCV_DiameterVert.InRearPosition AND
    Cylinder.List.fbUpCV_DiameterClamp.InRearPosition AND
    Cylinder.List.fbStackPush.InRearPosition AND
    Cylinder.List.fbLowCV_Press1.InRearPosition AND
    Cylinder.List.fbLowCV_Press2.InRearPosition AND
    Cylinder.List.fbLowCV_Press3.InRearPosition AND
    Cylinder.List.fbLowCV_Press4.InRearPosition AND
    Cylinder.List.fbLowCV_Block1.InRearPosition AND
    Cylinder.List.fbLowCV_Block2.InRearPosition;
END_METHOD

METHOD M_CheckStorageMotorInStop : BOOL
VAR_INPUT
END_VAR
M_CheckStorageMotorInStop := Motor.List.LowCV.InStopped AND
    Motor.List.UpCV.InStopped AND
    Motor.List.WareHouseCV_01.InStopped AND
    Motor.List.WareHouseCV_02.InStopped AND
    Motor.List.WareHouseCV_03.InStopped AND
    Motor.List.WareHouseCV_04.InStopped AND
    Motor.List.WareHouseCV_05.InStopped AND
    Motor.List.WareHouseCV_06.InStopped AND
    Motor.List.WareHouseCV_07.InStopped AND
    Motor.List.WareHouseCV_08.InStopped AND
    Motor.List.WareHouseCV_09.InStopped AND
    Motor.List.WareHouseCV_10.InStopped AND
    Motor.List.WareHouseCV_11.InStopped AND
    Motor.List.WareHouseCV_12.InStopped AND
    Motor.List.WareHouseCV_13.InStopped AND
    Motor.List.WareHouseCV_14.InStopped AND
    Motor.List.WareHouseCV_15.InStopped AND
    Motor.List.WareHouseCV_16.InStopped AND
    Motor.List.WareHouseCV_17.InStopped AND
    Motor.List.WareHouseCV_18.InStopped AND
    Motor.List.WareHouseCV_19.InStopped AND
    Motor.List.WareHouseCV_20.InStopped;
END_METHOD

METHOD M_GetErrorMsg : T_MaxString
VAR_INPUT
	xErrorID: INT;
END_VAR

VAR
	
END_VAR
CASE xErrorID OF
    0:
        M_GetErrorMsg := 'No Error';
    1:
        M_GetErrorMsg := 'FB_StorageHoming ErrorID 1: Action time out';
    2:
        M_GetErrorMsg := 'FB_StorageHoming ErrorID 2: Cylinder not ready';
    3:
        M_GetErrorMsg := 'FB_StorageHoming ErrorID 3: Motor not ready';
    4:
		M_GetErrorMsg := 'FB_StorageHoming ErrorID 4: FanucRobot can not homing';
	10:
		M_GetErrorMsg := 'FB_StorageHoming ErrorID 10: Storage FanucRobot FeedOut to NG Conveyor not busy';
	11:
		M_GetErrorMsg := 'FB_StorageHoming ErrorID 11: Storage FanucRobot FeedOut to NG Conveyor Done Timeout';
END_CASE
END_METHOD

METHOD M_RetractStorageCylinder : BOOL
VAR_INPUT
END_VAR
Cylinder.List.fbUpCV_FeedInPress1.M_Retract();
Cylinder.List.fbUpCV_FeedInPress2.M_Retract();
Cylinder.List.fbUpCV_DiameterPress.M_Retract();
Cylinder.List.fbUpCV_CamaraPress1.M_Retract();
Cylinder.List.fbUpCV_CamaraPress2.M_Retract();
Cylinder.List.fbUpCV_CamaraPress3.M_Retract();
Cylinder.List.fbUpCV_CamaraPress4.M_Retract();
Cylinder.List.fbUpCV_Block1.M_Retract();
Cylinder.List.fbUpCV_Block2.M_Retract();
Cylinder.List.fbUpCV_Block3.M_Retract();
Cylinder.List.fbUpCV_DiameterHoriz.M_Retract();
Cylinder.List.fbUpCV_DiameterVert.M_Retract();
Cylinder.List.fbUpCV_DiameterClamp.M_Retract();
Cylinder.List.fbStackPush.M_Retract();
Cylinder.List.fbLowCV_Press1.M_Retract();
Cylinder.List.fbLowCV_Press2.M_Retract();
Cylinder.List.fbLowCV_Press3.M_Retract();
Cylinder.List.fbLowCV_Press4.M_Retract();
Cylinder.List.fbLowCV_Block1.M_Retract();
Cylinder.List.fbLowCV_Block2.M_Retract();

M_RetractStorageCylinder := TRUE;
END_METHOD

METHOD M_StopStorageMotor : BOOL
VAR_INPUT
END_VAR
Motor.List.LowCV.M_MotorStop();
Motor.List.UpCV.M_MotorStop();
Motor.List.WareHouseCV_01.M_MotorStop();
Motor.List.WareHouseCV_02.M_MotorStop();
Motor.List.WareHouseCV_03.M_MotorStop();
Motor.List.WareHouseCV_04.M_MotorStop();
Motor.List.WareHouseCV_05.M_MotorStop();
Motor.List.WareHouseCV_06.M_MotorStop();
Motor.List.WareHouseCV_07.M_MotorStop();
Motor.List.WareHouseCV_08.M_MotorStop();
Motor.List.WareHouseCV_09.M_MotorStop();
Motor.List.WareHouseCV_10.M_MotorStop();
Motor.List.WareHouseCV_11.M_MotorStop();
Motor.List.WareHouseCV_12.M_MotorStop();
Motor.List.WareHouseCV_13.M_MotorStop();
Motor.List.WareHouseCV_14.M_MotorStop();
Motor.List.WareHouseCV_15.M_MotorStop();
Motor.List.WareHouseCV_16.M_MotorStop();
Motor.List.WareHouseCV_17.M_MotorStop();
Motor.List.WareHouseCV_18.M_MotorStop();
Motor.List.WareHouseCV_19.M_MotorStop();
Motor.List.WareHouseCV_20.M_MotorStop();

M_StopStorageMotor := TRUE;
END_METHOD

METHOD ResetAction
VAR_OUTPUT
    xComplete : BOOL := TRUE;
END_VAR
uiStorageHomingStep := 0;
RobotResetCMD := FALSE;
CylinderCheckTon.IN := FALSE;
MotorCheckTon.IN := FALSE;
FanucRobotCheckTon.IN := FALSE;
RackMotorHomeRequest := FALSE;

_fbRobotRegionMove_FeedInConveyor.M_ResetHomingFeedOut();

TON_RobotFeedOutCommand.IN  := FALSE;
TON_RobotTimeOut.IN			:= FALSE;
tonPowerCycle.IN			:= FALSE;
tonPowerCycleTimeout.IN		:= FALSE;
tonStartupDelay.IN			:= FALSE;
END_METHOD

METHOD StartAction
VAR_OUTPUT
    xComplete : BOOL := TRUE;
	iErrorID : INT := 0;
END_VAR

VAR
	uiCylinderIndex :UINT;
	uiMotorIndex : UINT;
END_VAR
Homed := FALSE;
RackMotorHomeRequest := false;
ResetRobotDelay.IN := FALSE;
uiStorageHomingStep := 0;

_fbRobotRegionMove_FeedInConveyor.M_ResetHomingFeedOut();

TON_RobotFeedOutCommand.IN  := FALSE;
TON_RobotTimeOut.IN			:= FALSE;
tonPowerCycle.IN			:= FALSE;
tonPowerCycleTimeout.IN		:= FALSE;
tonStartupDelay.IN			:= FALSE;

IF service.AutoMode_RobotRegionMove_FeedInConveyor.Command.Execute OR
	service.AutoMode_RobotRegionMove_FeedInConveyor.Status.Busy OR 
	service.AutoMode_RobotRegionMove_FeedInConveyor.Status.Error OR
	 service.AutoMode_RobotAbsMove.HandShake.Execute OR  
	 service.AutoMode_RobotAbsMove.HandShake.Busy OR 
	 service.AutoMode_RobotAbsMove.HandShake.Error
THEN
	iErrorID := 20;
ELSE
	xComplete := TRUE;
END_IF
END_METHOD

END_FUNCTION_BLOCK

// ---- Library/20_MachineUnits/21_StorageArea/Service/FB_DiameterMovement.TcPOU
FUNCTION_BLOCK FB_DiameterMovement EXTENDS FB_ObjectBase_V2
VAR_INPUT
//    Execute    :BOOL;   // True : This prog will start.
//    Abort      :BOOL;   // True : This prog will be abort.
//    Reset      :BOOL;   // True : This prog will be reset.
//    ObjectName :STRING; // Set this fb name(About it's action)
	
	bContinue:BOOL;
	
//	DiameterHorizontalCylinder 	:REFERENCE TO FB_Cylinder;	//測徑橫移氣壓缸
//	DiameterUpDownCylinder		:REFERENCE TO FB_Cylinder;	//測徑上下氣壓缸
//	DiameterClampCylinder		:REFERENCE TO FB_Cylinder; //測徑夾爪氣壓缸

	Cylinder : REFERENCE TO UNI_CylinderList;
	
END_VAR

VAR_OUTPUT
//    Busy    :BOOL;        // True : This prog is running.
//    Done    :BOOL;        // True : Command has been executed.
//    Aborted :BOOL;        // True : This prog is aborted.
//    Error   :BOOL;        // True : This prog has an error.
//    ErrorID :UINT;       // Output ErrorID
//    Status  :T_MaxString; // Output this prog status by string(255bytes)
	PickDone	:BOOL;
END_VAR

VAR
//    eState :E_MethodStatus_Basic;
//	uiExecutingStep : UDINT; // This var is used to been controll STATE_EXECUTING process.
//	uiResettingStep : UDINT;
//	uiAbortingStep : UDINT;
//	_Executed :BOOL; // Executing process completed.
//	_Error : BOOL; // FB has an error.
//	_ResetCompleted : BOOL; // FB resetting completed.
//	_AbortCompleted : BOOL; // FB aborting completed.
//	_Abort		: BOOL;
	strStatus	: STRING;
	uiResumeStep : UINT;
	tonDiameterTimeoutTwo :TON;
	
END_VAR

A00_BasicUnits();
SUPER^.A10_StateControl();

ACTION A00_BasicUnits:
tonDiameterTimeoutTwo(PT:=T#2S);
END_ACTION

METHOD GetModelState
VAR_OUTPUT
    xDone    :BOOL;
    xBusy    :BOOL;
    xError   :BOOL;
    xAborted :BOOL;
    iErrorID :UDINT;
	UniqueErrorCode : STRING;
END_VAR
xDone    := Done;
xBusy    := Busy;
xError   := Error;
xAborted := Abort;
iErrorID := ErrorID;
END_METHOD

METHOD GetName : STRING
GetName := ObjectName;
END_METHOD

METHOD  M_STATE_ABORTED
VAR_INPUT
END_VAR
ERROR :=TRUE;
Status := strStatus;

IF NOT Execute THEN
	eSTATE:=STATE_RESETTING;
END_IF

IF Execute AND Reset THEN
	uiExecutingStep :=uiResumeStep;
	eSTATE:=STATE_EXECUTING;
END_IF
END_METHOD

METHOD  M_STATE_ABORTING
VAR_INPUT
END_VAR
CASE uiAbortingStep OF
	
	
	9999:	_AbortCompleted:=TRUE;
END_CASE

IF _AbortCompleted THEN	
	eSTATE :=STATE_ABORTED;
END_IF
END_METHOD

METHOD  M_STATE_DONE
VAR_INPUT
END_VAR
Busy := FALSE;
Done:=TRUE;

IF NOT Execute THEN
	eSTATE:=STATE_RESETTING;
END_IF
END_METHOD

METHOD  M_STATE_DORMANT
VAR_INPUT
END_VAR
_Executed:=FALSE;
_Error	:=FALSE;
_Abort :=FALSE;
strStatus :='FB_DiameterMovement: No Error';
uiResettingStep:=0;
uiExecutingStep :=0;
tonDiameterTimeoutTwo.IN:=FALSE;
Error := Busy := Done := FALSE;

IF Execute THEN
	eSTATE:=STATE_EXECUTING;
END_IF
END_METHOD

METHOD  M_STATE_ERROR
VAR_INPUT
END_VAR
ERROR :=TRUE;
Busy :=FALSE;
Done := FALSE;
Status := strStatus;
IF NOT Execute THEN	
eSTATE:=STATE_RESETTING;
END_IF
END_METHOD

METHOD  M_STATE_EXECUTING
VAR_INPUT
END_VAR
Busy :=TRUE;

CASE uiExecutingStep OF
	

0: //Standby todo : check 
	
		uiExecutingStep:=10;
10:
		
		IF Cylinder.List.fbUpCV_DiameterHoriz.xError THEN
			Cylinder.List.fbUpCV_DiameterHoriz.M_Reset();
		END_IF
		IF Cylinder.List.fbUpCV_DiameterVert.xError THEN
			Cylinder.List.fbUpCV_DiameterVert.M_Reset();
		END_IF
		IF Cylinder.List.fbUpCV_DiameterClamp.xError THEN
			Cylinder.List.fbUpCV_DiameterClamp.M_Reset();
		END_IF
		uiExecutingStep:=20;
		
20:
	Cylinder.List.fbUpCV_DiameterVert.M_Retract();
	IF Cylinder.List.fbUpCV_DiameterClamp.InFrontPosition THEN
		uiExecutingStep:=30;
	ELSE
		uiExecutingStep:=60;	
	END_IF
30:
	
	IF Cylinder.List.fbUpCV_DiameterVert.InRearPosition THEN
		Cylinder.List.fbUpCV_DiameterHoriz.M_Extend();
		uiExecutingStep:=40;
	END_IF
40:		
	IF Cylinder.List.fbUpCV_DiameterHoriz.InFrontPosition THEN
		Cylinder.List.fbUpCV_DiameterClamp.M_Retract();
		uiExecutingStep:=50;
	END_IF
50:	
	IF Cylinder.List.fbUpCV_DiameterClamp.InRearPosition THEN
		uiExecutingStep:=60;
	END_IF
	
60 : 
	Cylinder.List.fbUpCV_DiameterHoriz.M_Retract();
		uiExecutingStep:=70;
70:
	IF Cylinder.List.fbUpCV_DiameterHoriz.InRearPosition THEN
		uiExecutingStep:=1000;	
	END_IF
			
	

1000:// Pick to diameter camera position start: Clamp down
	Cylinder.List.fbUpCV_DiameterVert.M_Extend();
	uiExecutingStep:=1100;
	
1100:// wait clamp down
	tonDiameterTimeoutTwo.IN:=TRUE;
	IF 	Cylinder.List.fbUpCV_DiameterVert.InFrontPosition THEN
		tonDiameterTimeoutTwo.IN:=FALSE;
		uiExecutingStep:=1200;
	END_IF
	IF tonDiameterTimeoutTwo.Q THEN
		_Error :=TRUE;
		strStatus:='FB_DiameterMovement Step 1100: Cylinder.List.fbUpCV_DiameterVert MoveForward Timeout';
	END_IF
	
1200: // Clamp close
	Cylinder.List.fbUpCV_DiameterClamp.M_Extend();
	uiExecutingStep:=1300;

1300://wait clamp close
	tonDiameterTimeoutTwo.IN:=TRUE;
	IF 	Cylinder.List.fbUpCV_DiameterClamp.InFrontPosition THEN
		tonDiameterTimeoutTwo.IN :=FALSE;
		uiExecutingStep:=1400;
	END_IF
	IF tonDiameterTimeoutTwo.Q THEN
		_Error :=TRUE;
		strStatus:='FB_DiameterMovement Step 1300: Cylinder.List.fbUpCV_DiameterClamp M_Extend Timeout';
	END_IF
1400 : //Clamp up
	Cylinder.List.fbUpCV_DiameterVert.M_Retract();
	uiExecutingStep:=1500;	

1500:// wait clamp up
		tonDiameterTimeoutTwo.IN :=TRUE;
	IF 	Cylinder.List.fbUpCV_DiameterVert.InRearPosition THEN
		tonDiameterTimeoutTwo.IN :=FALSE;
		uiExecutingStep:=1600;
	END_IF
	IF tonDiameterTimeoutTwo.Q THEN
		_Error :=TRUE;
		strStatus:='FB_DiameterMovement Step 1500: Cylinder.List.fbUpCV_DiameterVert M_Retract Timeout';
	END_IF
1600: //Move horizontal
	Cylinder.List.fbUpCV_DiameterHoriz.M_Extend();
	uiExecutingStep:=1700;

1700://wait move horizontal
		tonDiameterTimeoutTwo.IN:=TRUE;
	IF 	Cylinder.List.fbUpCV_DiameterHoriz.InFrontPosition THEN
		tonDiameterTimeoutTwo.IN :=FALSE;
		uiExecutingStep:=1800;
	END_IF
		IF tonDiameterTimeoutTwo.Q THEN
		_Error :=TRUE;
		strStatus:='FB_DiameterMovement Step 1700: Cylinder.List.fbUpCV_DiameterHoriz M_Extend Timeout';
	END_IF

1800://Move down to diameter camera position
	Cylinder.List.fbUpCV_DiameterVert.M_Extend();
	uiExecutingStep:=1900;
	
1900:
		tonDiameterTimeoutTwo.IN:=TRUE;
	IF 	Cylinder.List.fbUpCV_DiameterVert.InFrontPosition THEN
		tonDiameterTimeoutTwo.IN :=FALSE;
		uiExecutingStep:=2000;
	END_IF
	IF tonDiameterTimeoutTwo.Q THEN
		_Error :=TRUE;
		strStatus:='FB_DiameterMovement Step 1900: Cylinder.List.fbUpCV_DiameterVert M_Extend Timeout';
	END_IF

2000: 
	PickDone :=TRUE;
	IF bContinue THEN
		PickDone :=FALSE;
		uiExecutingStep:=5000;
	END_IF

5000: // Place needle back to box start
	Cylinder.List.fbUpCV_DiameterVert.M_Retract();
	uiExecutingStep:=5100;
	
5100:// wait clamp down
	tonDiameterTimeoutTwo.IN :=TRUE;
	IF 	Cylinder.List.fbUpCV_DiameterVert.InRearPosition THEN
		tonDiameterTimeoutTwo.IN :=FALSE;
		uiExecutingStep:=5200;
	END_IF
	IF tonDiameterTimeoutTwo.Q THEN
		_Error :=TRUE;
		strStatus:='FB_DiameterMovement Step 5100: Cylinder.List.fbUpCV_DiameterVert M_Retract Timeout';
	END_IF
	
5200: 
		Cylinder.List.fbUpCV_DiameterHoriz.M_Retract();
		uiExecutingStep := 5300;

5300:
		tonDiameterTimeoutTwo.IN :=TRUE;
		IF Cylinder.List.fbUpCV_DiameterHoriz.InRearPosition THEN
			tonDiameterTimeoutTwo.IN :=FALSE;
			uiExecutingStep := 5400;
		END_IF
		IF tonDiameterTimeoutTwo.Q THEN
		_Error :=TRUE;
		strStatus:='FB_DiameterMovement Step 5300: Cylinder.List.fbUpCV_DiameterHoriz M_Retract Timeout';
		END_IF
5400 : 
		Cylinder.List.fbUpCV_DiameterVert.M_Extend();
		uiExecutingStep:=5500;

5500:
		tonDiameterTimeoutTwo.IN :=TRUE;
		IF 	Cylinder.List.fbUpCV_DiameterVert.InFrontPosition THEN
			tonDiameterTimeoutTwo.IN:=FALSE;
			uiExecutingStep:=5600;
		END_IF
		IF tonDiameterTimeoutTwo.Q THEN
		_Error :=TRUE;
		strStatus:='FB_DiameterMovement Step 5500: Cylinder.List.fbUpCV_DiameterVert M_Extend Timeout';
		END_IF
5600: 
		Cylinder.List.fbUpCV_DiameterClamp.M_Retract();
		uiExecutingStep := 5700;
5700:	
		tonDiameterTimeoutTwo.IN :=TRUE;
		IF Cylinder.List.fbUpCV_DiameterClamp.InRearPosition THEN
			tonDiameterTimeoutTwo.IN :=FALSE;
			uiExecutingStep :=5800;
		END_IF
		IF tonDiameterTimeoutTwo.Q THEN
		_Error :=TRUE;
		strStatus:='FB_DiameterMovement Step 5700: Cylinder.List.fbUpCV_DiameterClamp M_Retract Timeout';
		END_IF
5800:
		Cylinder.List.fbUpCV_DiameterVert.M_Retract();
		 uiExecutingStep := 5900;
5900:
		tonDiameterTimeoutTwo.IN :=TRUE;
		IF Cylinder.List.fbUpCV_DiameterVert.InRearPosition THEN
			tonDiameterTimeoutTwo.IN :=FALSE;
		uiExecutingStep :=6000;
		END_IF
		IF tonDiameterTimeoutTwo.Q THEN
		_Error :=TRUE;
		strStatus:='FB_DiameterMovement Step 5900: Cylinder.List.fbUpCV_DiameterVert M_Retract Timeout';
		END_IF
6000:
		_Executed:= TRUE;





END_CASE
	
IF NOT Execute THEN
	eState:=STATE_RESETTING;
END_IF
IF _Error THEN
	eState:=STATE_ERROR;
END_IF
IF _Abort THEN
	eSTATE:=STATE_ABORTING;
END_IF
IF _Executed THEN
	eSTATE:=STATE_Done;
END_IF
END_METHOD

METHOD  M_STATE_RESETTING
VAR_INPUT
END_VAR
Error :=FALSE;
Busy := FALSE;


CASE uiResettingStep OF
	0 : 
		
		IF Cylinder.List.fbUpCV_DiameterHoriz.xError THEN
			Cylinder.List.fbUpCV_DiameterHoriz.M_Reset();
		END_IF
		IF Cylinder.List.fbUpCV_DiameterVert.xError THEN
			Cylinder.List.fbUpCV_DiameterVert.M_Reset();
		END_IF
		IF Cylinder.List.fbUpCV_DiameterClamp.xError THEN
			Cylinder.List.fbUpCV_DiameterClamp.M_Reset();
		END_IF
		uiResettingStep:=100;
		
	100:
		Cylinder.List.fbUpCV_DiameterVert.M_Retract();
		IF Cylinder.List.fbUpCV_DiameterClamp.InFrontPosition THEN
			uiResettingStep:=1000;
		ELSE
			uiResettingStep:=2000;	
		END_IF
	1000:
			
			IF Cylinder.List.fbUpCV_DiameterVert.InRearPosition THEN
				Cylinder.List.fbUpCV_DiameterHoriz.M_Extend();
				uiResettingStep:=1200;
			END_IF
	1200:		
			IF Cylinder.List.fbUpCV_DiameterHoriz.InFrontPosition THEN
				Cylinder.List.fbUpCV_DiameterClamp.M_Retract();
				uiResettingStep:=1300;
			END_IF
	1300:	
			IF Cylinder.List.fbUpCV_DiameterClamp.InRearPosition THEN
				uiResettingStep:=2000;
			END_IF
		
	2000 : 
			Cylinder.List.fbUpCV_DiameterHoriz.M_Retract();
				uiResettingStep:=2100;
	2100:
			IF Cylinder.List.fbUpCV_DiameterHoriz.InRearPosition THEN
				uiResettingStep:=9999;	
			END_IF
			
	9999:
		_ResetCompleted:=TRUE;
END_CASE
IF _ResetCompleted THEN
	eSTATE:=STATE_DORMANT;
END_IF
END_METHOD

END_FUNCTION_BLOCK

// ---- Library/20_MachineUnits/21_StorageArea/Service/FB_UpperFeedInConveyor.TcPOU
FUNCTION_BLOCK FB_UpperFeedInConveyor EXTENDS FB_ObjectBase_V2
VAR_INPUT
	
	_fbDiameterMovement : REFERENCE TO FB_DiameterMovement;
	
	Cylinder 	: REFERENCE TO UNI_CylinderList;
	Motor	 	: REFERENCE TO UNI_MotorList;
	Input 	 	: REFERENCE TO ST_InputTable;
	OutPut	 	: REFERENCE TO ST_OutputTable;
	
	Info		: ST_Auto_UpperFeedInConveyorInfo;

	AddingBox	: BOOL;
//	Pause		: BOOL;	// True: 暫停機台動作和計時器

//    Execute    :BOOL;   // True : This prog will start.
//    Abort      :BOOL;   // True : This prog will be abort.
//    Reset      :BOOL;   // True : This prog will be reset.
//    ObjectName :STRING; // Set this fb name(About it's action)
END_VAR

VAR_OUTPUT
//	Status		: ST_StatusBasic;
	FeedBack    : ST_Auto_UpperFeedInConveyorFeedback;
	_bForceUpperCV_Use	: BOOL;
//	Paused		: BOOL;	// True: 目前處於暫停狀態	
//    Busy    :BOOL;        // True : This prog is running.
//    Done    :BOOL;        // True : Command has been executed.
//    Aborted :BOOL;        // True : This prog is aborted.
//    Error   :BOOL;        // True : This prog has an error.
//    ErrorID :UINT;       // Output ErrorID
//    Status  :T_MaxString; // Output this prog status by string(255bytes)
	RobotService_CheckUPCVServicedone	: BOOL;
END_VAR

VAR
//    eState :E_MethodStatus_Basic;
//	uiExecutingStep : UDINT; // This var is used to been controll STATE_EXECUTING process.
//	uiResettingStep : UDINT;
//	uiAbortingStep : UDINT;
//	_Executed :BOOL; // Executing process completed.
//	_Error : BOOL; // FB has an error.
//	_ResetCompleted : BOOL; // FB resetting completed.
//	_AbortCompleted : BOOL; // FB aborting completed.
	//_Abort		: BOOL;
	strStatus	: T_MaxString;
	uiResumeStep : UINT;
	iMoveConveyor	:INT;// 1 = MoveForward , -1 = Move reverse , 0 or other = Stop
	tonUpperConveyorTimeOut			:TON;
	tonUpperConveyorDelay			:TON;
	tonUpperTimeOut					:TON;
	tonUpperTimeOutFive 			:TON;
	tonWaitSecondBoxArriveTimeout 	:TON;
	tonFeedAirBlowtime 				:TON;
	tonReverseConveyorDelay			:TON;
	TON_CheckHaveBox				:TON ;
	NoFirstBoxDiameter : BOOL;
	SecondBox	:BOOL;
	bSecondBoxInCameraPos :BOOL;
	uiFirstBoxDiameterStep :UINT :=0;
	uiSecondBoxAirBlowStep :UINT :=0;
	_UniqueErrorCode :STRING;
	
	
	//record time for C# photo
	tRecordTimer 		: ARRAY [1..100] OF TIME;
	tRecordFirstTimer	: ARRAY [1..100] OF TIME;
	tRecordSecondTimer	: ARRAY [1..100] OF TIME;
	TON_RecordTimer 	: TON;
	TON_RecordFirstTimer		: TON ;
	TON_RecordSecondTimer		: TON;
	TSaveTime					: TIME;
	TSaveFirstTime				: TIME;
	TSaveSecondTime				: TIME;
	iArrayNumber 				: INT :=1;
	iResetNumber				: INT;
	bResetRecordInfo			: BOOL;

	// ===== 暫停功能相關變數 =====
	_bPaused					: BOOL;
	_bPauseEdge					: BOOL;	// 邊緣檢測

	// 記住計時器原本 IN 狀態
	bWasActive_UpperConveyorTimeOut			: BOOL;
	bWasActive_UpperConveyorDelay			: BOOL;
	bWasActive_UpperTimeOut					: BOOL;
	bWasActive_UpperTimeOutFive				: BOOL;
	bWasActive_WaitSecondBoxArriveTimeout	: BOOL;
	bWasActive_FeedAirBlowtime				: BOOL;
	bWasActive_ReverseConveyorDelay			: BOOL;
	bWasActive_CheckHaveBox					: BOOL;

	// 記住馬達/輸出狀態
	iSaved_MoveConveyor		: INT;
	bSaved_CamaraBlow		: BOOL;

	// 計時器剩餘時間 (恢復後使用)
	tRemaining_UpperConveyorTimeOut			: TIME;
	tRemaining_UpperConveyorDelay			: TIME;
	tRemaining_UpperTimeOut					: TIME;
	tRemaining_UpperTimeOutFive				: TIME;
	tRemaining_WaitSecondBoxArriveTimeout	: TIME;
	tRemaining_FeedAirBlowtime				: TIME;
	tRemaining_ReverseConveyorDelay			: TIME;
	tRemaining_CheckHaveBox					: TIME;

	// 標記是否需要使用調整後的 PT
	bUseAdjustedPT_UpperConveyorTimeOut			: BOOL;
	bUseAdjustedPT_UpperConveyorDelay			: BOOL;
	bUseAdjustedPT_UpperTimeOut					: BOOL;
	bUseAdjustedPT_UpperTimeOutFive				: BOOL;
	bUseAdjustedPT_WaitSecondBoxArriveTimeout	: BOOL;
	bUseAdjustedPT_FeedAirBlowtime				: BOOL;
	bUseAdjustedPT_ReverseConveyorDelay			: BOOL;
	bUseAdjustedPT_CheckHaveBox					: BOOL;

END_VAR

A00_BasicUnits();
A01_PauseControl();	// 暫停控制

// 暫停時不執行狀態機
IF NOT _bPaused THEN
	SUPER^.A10_StateControl();
END_IF

ACTION A00_BasicUnits:
// 計時器調用 - 根據暫停恢復標志決定 PT 值
// 當計時器 IN=FALSE 時，清除標志並恢復原始 PT

// tonUpperConveyorTimeOut
IF bUseAdjustedPT_UpperConveyorTimeOut THEN
	tonUpperConveyorTimeOut(PT := tRemaining_UpperConveyorTimeOut);
	IF NOT tonUpperConveyorTimeOut.IN THEN
		bUseAdjustedPT_UpperConveyorTimeOut := FALSE;
	END_IF
ELSE
	tonUpperConveyorTimeOut(PT := T#20S);
END_IF

// tonUpperConveyorDelay (PT 由外部設定)
IF bUseAdjustedPT_UpperConveyorDelay THEN
	tonUpperConveyorDelay(PT := tRemaining_UpperConveyorDelay);
	IF NOT tonUpperConveyorDelay.IN THEN
		bUseAdjustedPT_UpperConveyorDelay := FALSE;
	END_IF
ELSE
	tonUpperConveyorDelay();
END_IF

// tonUpperTimeOut
IF bUseAdjustedPT_UpperTimeOut THEN
	tonUpperTimeOut(PT := tRemaining_UpperTimeOut);
	IF NOT tonUpperTimeOut.IN THEN
		bUseAdjustedPT_UpperTimeOut := FALSE;
	END_IF
ELSE
	tonUpperTimeOut(PT := T#5S);
END_IF

// tonUpperTimeOutFive
IF bUseAdjustedPT_UpperTimeOutFive THEN
	tonUpperTimeOutFive(PT := tRemaining_UpperTimeOutFive);
	IF NOT tonUpperTimeOutFive.IN THEN
		bUseAdjustedPT_UpperTimeOutFive := FALSE;
	END_IF
ELSE
	tonUpperTimeOutFive(PT := T#60S);
END_IF

// tonWaitSecondBoxArriveTimeout
IF bUseAdjustedPT_WaitSecondBoxArriveTimeout THEN
	tonWaitSecondBoxArriveTimeout(PT := tRemaining_WaitSecondBoxArriveTimeout);
	IF NOT tonWaitSecondBoxArriveTimeout.IN THEN
		bUseAdjustedPT_WaitSecondBoxArriveTimeout := FALSE;
	END_IF
ELSE
	tonWaitSecondBoxArriveTimeout(PT := T#20S);
END_IF

// tonFeedAirBlowtime
IF bUseAdjustedPT_FeedAirBlowtime THEN
	tonFeedAirBlowtime(PT := tRemaining_FeedAirBlowtime);
	IF NOT tonFeedAirBlowtime.IN THEN
		bUseAdjustedPT_FeedAirBlowtime := FALSE;
	END_IF
ELSE
	tonFeedAirBlowtime(PT := Info.FeedAirblowTime);
END_IF

// tonReverseConveyorDelay
IF bUseAdjustedPT_ReverseConveyorDelay THEN
	tonReverseConveyorDelay(PT := tRemaining_ReverseConveyorDelay);
	IF NOT tonReverseConveyorDelay.IN THEN
		bUseAdjustedPT_ReverseConveyorDelay := FALSE;
	END_IF
ELSE
	tonReverseConveyorDelay(PT := T#6S);
END_IF

// TON_CheckHaveBox
IF bUseAdjustedPT_CheckHaveBox THEN
	TON_CheckHaveBox(PT := tRemaining_CheckHaveBox);
	IF NOT TON_CheckHaveBox.IN THEN
		bUseAdjustedPT_CheckHaveBox := FALSE;
	END_IF
ELSE
	TON_CheckHaveBox(PT := T#35S);
END_IF

ErrorID := 2710;

TON_RecordTimer(PT := T#1D);
TON_RecordFirstTimer(PT := T#1D);
TON_RecordSecondTimer(PT := T#1D);

IF bResetRecordInfo THEN
	FOR iResetNumber := 1 TO 100 DO
		tRecordTimer[iResetNumber] := T#0S;
		tRecordFirstTimer[iResetNumber] := T#0S;
		tRecordSecondTimer[iResetNumber] := T#0S;
	END_FOR
END_IF
END_ACTION

ACTION A01_PauseControl:
// A01_PauseControl - 暫停控制邏輯

Paused := _bPaused;

// 只在執行狀態處理暫停
IF eState <> STATE_EXECUTING THEN
	_bPaused := FALSE;
	RETURN;
END_IF

// ===== 進入暫停 (上升邊緣) =====
IF Pause AND NOT _bPauseEdge THEN
	_bPauseEdge := TRUE;

	IF NOT _bPaused THEN
		_bPaused := TRUE;

		// 保存計時器活動狀態和剩餘時間
		bWasActive_UpperConveyorTimeOut := tonUpperConveyorTimeOut.IN;
		tRemaining_UpperConveyorTimeOut := T#20S - tonUpperConveyorTimeOut.ET;

		bWasActive_UpperConveyorDelay := tonUpperConveyorDelay.IN;
		tRemaining_UpperConveyorDelay := tonUpperConveyorDelay.PT - tonUpperConveyorDelay.ET;

		bWasActive_UpperTimeOut := tonUpperTimeOut.IN;
		tRemaining_UpperTimeOut := T#5S - tonUpperTimeOut.ET;

		bWasActive_UpperTimeOutFive := tonUpperTimeOutFive.IN;
		tRemaining_UpperTimeOutFive := T#60S - tonUpperTimeOutFive.ET;

		bWasActive_WaitSecondBoxArriveTimeout := tonWaitSecondBoxArriveTimeout.IN;
		tRemaining_WaitSecondBoxArriveTimeout := T#20S - tonWaitSecondBoxArriveTimeout.ET;

		bWasActive_FeedAirBlowtime := tonFeedAirBlowtime.IN;
		tRemaining_FeedAirBlowtime := Info.FeedAirblowTime - tonFeedAirBlowtime.ET;

		bWasActive_ReverseConveyorDelay := tonReverseConveyorDelay.IN;
		tRemaining_ReverseConveyorDelay := T#6S - tonReverseConveyorDelay.ET;

		bWasActive_CheckHaveBox := TON_CheckHaveBox.IN;
		tRemaining_CheckHaveBox := T#35S - TON_CheckHaveBox.ET;

		// 保存馬達狀態
		iSaved_MoveConveyor := iMoveConveyor;
		bSaved_CamaraBlow := OutPut.bCamara_Blow;

		// 停止所有計時器
		tonUpperConveyorTimeOut.IN := FALSE;
		tonUpperConveyorDelay.IN := FALSE;
		tonUpperTimeOut.IN := FALSE;
		tonUpperTimeOutFive.IN := FALSE;
		tonWaitSecondBoxArriveTimeout.IN := FALSE;
		tonFeedAirBlowtime.IN := FALSE;
		tonReverseConveyorDelay.IN := FALSE;
		TON_CheckHaveBox.IN := FALSE;

		// 停止馬達
		iMoveConveyor := 0;
		Motor.list.UpCV.M_MotorStop();

		// 停止輸出
		OutPut.bCamara_Blow := FALSE;
	END_IF
END_IF

// ===== 離開暫停 (下降邊緣) =====
IF NOT Pause AND _bPauseEdge AND GVL_ADS.OpPannel_Status.StartBtnStatus THEN
	_bPauseEdge := FALSE;

	IF _bPaused THEN
		_bPaused := FALSE;

		// 恢復馬達狀態
		iMoveConveyor := iSaved_MoveConveyor;
		OutPut.bCamara_Blow := bSaved_CamaraBlow;

		// 設置標志：需要使用調整後的 PT
		IF bWasActive_UpperConveyorTimeOut THEN
			bUseAdjustedPT_UpperConveyorTimeOut := TRUE;
			tonUpperConveyorTimeOut.IN := TRUE;
		END_IF

		IF bWasActive_UpperConveyorDelay THEN
			bUseAdjustedPT_UpperConveyorDelay := TRUE;
			tonUpperConveyorDelay.IN := TRUE;
		END_IF

		IF bWasActive_UpperTimeOut THEN
			bUseAdjustedPT_UpperTimeOut := TRUE;
			tonUpperTimeOut.IN := TRUE;
		END_IF

		IF bWasActive_UpperTimeOutFive THEN
			bUseAdjustedPT_UpperTimeOutFive := TRUE;
			tonUpperTimeOutFive.IN := TRUE;
		END_IF

		IF bWasActive_WaitSecondBoxArriveTimeout THEN
			bUseAdjustedPT_WaitSecondBoxArriveTimeout := TRUE;
			tonWaitSecondBoxArriveTimeout.IN := TRUE;
		END_IF

		IF bWasActive_FeedAirBlowtime THEN
			bUseAdjustedPT_FeedAirBlowtime := TRUE;
			tonFeedAirBlowtime.IN := TRUE;
		END_IF

		IF bWasActive_ReverseConveyorDelay THEN
			bUseAdjustedPT_ReverseConveyorDelay := TRUE;
			tonReverseConveyorDelay.IN := TRUE;
		END_IF

		IF bWasActive_CheckHaveBox THEN
			bUseAdjustedPT_CheckHaveBox := TRUE;
			TON_CheckHaveBox.IN := TRUE;
		END_IF
	END_IF
END_IF
END_ACTION

METHOD GetModelState
VAR_OUTPUT
    xDone    :BOOL;
    xBusy    :BOOL;
    xError   :BOOL;
    xAborted :BOOL;
    iErrorID :UDINT;
	UniqueErrorCode : STRING;
END_VAR
xDone    := Done;
xBusy    := Busy;
xError   := Error;
xAborted := Abort;
iErrorID := ErrorID;
END_METHOD

METHOD GetName : STRING
GetName := ObjectName;
END_METHOD

METHOD  M_STATE_ABORTED
VAR_INPUT
END_VAR
ERROR	:= TRUE;
Busy	:= FALSE;
Aborted	:= TRUE;
_Abort	:= FALSE;
UniqueErrorCode	:=_UniqueErrorCode;
SUPER^.Status	:= strStatus;
uiAbortingStep	:= 0;
_AbortCompleted := FALSE;

IF NOT Execute THEN
	eSTATE:=STATE_RESETTING;
	
ELSIF Execute AND Reset THEN

		CASE uiExecutingStep OF
			
			460:	//Box1 done step abort
				uiExecutingStep :=450;
				strStatus :='FB_UpperFeedInConveyor Step 460: Check FirstBoxCamaraDone info retry';
			
				
		END_CASE
	
	error 	:= FALSE;	
	Aborted := FALSE;
	eSTATE	:= STATE_EXECUTING;
	
END_IF
END_METHOD

METHOD  M_STATE_ABORTING
VAR_INPUT
END_VAR
Busy :=FALSE;
CASE uiAbortingStep OF
	0:
		tonUpperConveyorTimeOut.IN 	:=FALSE;
		tonUpperConveyorDelay.IN	:=FALSE;
		tonUpperTimeOut.IN 			:=FALSE;
		tonUpperTimeOutfive.IN		:=FALSE;
		TON_CheckHaveBox.IN 		:=FALSE;
		uiAbortingStep :=100;
	100:
		Motor.List.UpCV.M_MotorStop();
		OutPut.bCamara_Blow :=FALSE;
		IF Motor.List.UpCV.InStopped THEN
			uiAbortingStep :=9999;
		END_IF
	9999:	
		_AbortCompleted:=TRUE;
END_CASE

IF _AbortCompleted THEN	
	eSTATE :=STATE_ABORTED;
END_IF
END_METHOD

METHOD  M_STATE_DONE
VAR_INPUT
END_VAR
Busy := FALSE;
Done:=TRUE;
_fbDiameterMovement.Execute := FALSE;
_fbDiameterMovement.bContinue:=FALSE;
RobotService_CheckUPCVServicedone := TRUE;
IF NOT Execute THEN
	eSTATE:=STATE_RESETTING;
END_IF
END_METHOD

